cart04_front_temp														:= F_Temperature(TT_04_01, TT_04_01_offset);
cart04_front_temp_error 												:= TT_04_01_error OR iCount[6] < 30;
cart04_back_temp														:= F_Temperature(TT_04_03, TT_04_03_offset);
cart04_back_temp_error 													:= TT_04_03_Error OR iCount[7] < 30;
cart04_temp_front_calc(Error:= TT_04_01_error, Temp:= cart04_front_temp, Low:= sorbent_low_temp, High:= sorbent_high_temp, Total:= rTempTotal, Counter:= iTempCount);
cart04_temp_back_calc(Error:= TT_04_03_Error, Temp:= cart04_back_temp, Low:= sorbent_low_temp, High:= sorbent_high_temp, Total:= rTempTotal, Counter:= iTempCount);

cart05_front_temp														:= F_Temperature(TT_05_01, TT_05_01_offset);
cart05_front_temp_error 												:= TT_05_01_error OR iCount[8] < 30;
cart05_back_temp														:= F_Temperature(TT_05_03, TT_05_03_offset);
cart05_back_temp_error 													:= TT_05_03_Error OR iCount[9] < 30;
cart05_temp_front_calc(Error:= TT_05_01_error, Temp:= cart05_front_temp, Low:= sorbent_low_temp, High:= sorbent_high_temp, Total:= rTempTotal, Counter:= iTempCount);
cart05_temp_back_calc(Error:= TT_05_03_Error, Temp:= cart05_back_temp, Low:= sorbent_low_temp, High:= sorbent_high_temp, Total:= rTempTotal, Counter:= iTempCount);

cart06_front_temp														:= F_Temperature(TT_06_01, TT_06_01_offset);
cart06_front_temp_error 												:= TT_06_01_error OR iCount[10] < 30;
cart06_back_temp														:= F_Temperature(TT_06_03, TT_06_03_offset);
cart06_back_temp_error 													:= TT_06_03_Error OR iCount[11] < 30;
cart06_temp_front_calc(Error:= TT_06_01_error, Temp:= cart06_front_temp, Low:= sorbent_low_temp, High:= sorbent_high_temp, Total:= rTempTotal, Counter:= iTempCount);
cart06_temp_back_calc(Error:= TT_06_03_Error, Temp:= cart06_back_temp, Low:= sorbent_low_temp, High:= sorbent_high_temp, Total:= rTempTotal, Counter:= iTempCount);

cart07_front_temp														:= F_Temperature(TT_07_01, TT_07_01_offset);
cart07_front_temp_error 												:= TT_07_01_error OR iCount[12] < 30;
cart07_back_temp														:= F_Temperature(TT_07_03, TT_07_03_offset);
cart07_back_temp_error 													:= TT_07_03_Error OR iCount[13] < 30;
cart07_temp_front_calc(Error:= TT_07_01_error, Temp:= cart07_front_temp, Low:= sorbent_low_temp, High:= sorbent_high_temp, Total:= rTempTotal, Counter:= iTempCount);
cart07_temp_back_calc(Error:= TT_07_03_Error, Temp:= cart07_back_temp, Low:= sorbent_low_temp, High:= sorbent_high_temp, Total:= rTempTotal, Counter:= iTempCount);

cart08_front_temp														:= F_Temperature(TT_08_01, TT_08_01_offset);
cart08_front_temp_error 												:= TT_08_01_error OR iCount[14] < 30;
cart08_back_temp														:= F_Temperature(TT_08_03, TT_08_03_offset);
cart08_back_temp_error 													:= TT_08_03_Error OR iCount[15] < 30;
cart08_temp_front_calc(Error:= TT_08_01_error, Temp:= cart08_front_temp, Low:= sorbent_low_temp, High:= sorbent_high_temp, Total:= rTempTotal, Counter:= iTempCount);
cart08_temp_back_calc(Error:= TT_08_03_Error, Temp:= cart08_back_temp, Low:= sorbent_low_temp, High:= sorbent_high_temp, Total:= rTempTotal, Counter:= iTempCount);

cart09_front_temp														:= F_Temperature(TT_09_01, TT_09_01_offset);
cart09_front_temp_error 												:= TT_09_01_error OR iCount[16] < 30;
cart09_back_temp														:= F_Temperature(TT_09_03, TT_09_03_offset);
cart09_back_temp_error 													:= TT_09_03_Error OR iCount[17] < 30;
cart09_temp_front_calc(Error:= TT_09_01_error, Temp:= cart09_front_temp, Low:= sorbent_low_temp, High:= sorbent_high_temp, Total:= rTempTotal, Counter:= iTempCount);
cart09_temp_back_calc(Error:= TT_09_03_Error, Temp:= cart09_back_temp, Low:= sorbent_low_temp, High:= sorbent_high_temp, Total:= rTempTotal, Counter:= iTempCount);

cart10_front_temp														:= F_Temperature(TT_10_01, TT_10_01_offset);
cart10_front_temp_error 												:= TT_10_01_error OR iCount[18] < 30;
cart10_back_temp														:= F_Temperature(TT_10_03, TT_10_03_offset);
cart10_back_temp_error 													:= TT_10_03_Error OR iCount[19] < 30;
cart10_temp_front_calc(Error:= TT_10_01_error, Temp:= cart10_front_temp, Low:= sorbent_low_temp, High:= sorbent_high_temp, Total:= rTempTotal, Counter:= iTempCount);
cart10_temp_back_calc(Error:= TT_10_03_Error, Temp:= cart10_back_temp, Low:= sorbent_low_temp, High:= sorbent_high_temp, Total:= rTempTotal, Counter:= iTempCount);

cart11_front_temp														:= F_Temperature(TT_11_01, TT_11_01_offset);
cart11_front_temp_error 												:= TT_11_01_error OR iCount[20] < 30;
cart11_back_temp														:= F_Temperature(TT_11_03, TT_11_03_offset);
cart11_back_temp_error 													:= TT_11_03_Error OR iCount[21] < 30;
cart11_temp_front_calc(Error:= TT_11_01_error, Temp:= cart11_front_temp, Low:= sorbent_low_temp, High:= sorbent_high_temp, Total:= rTempTotal, Counter:= iTempCount);
cart11_temp_back_calc(Error:= TT_11_03_Error, Temp:= cart11_back_temp, Low:= sorbent_low_temp, High:= sorbent_high_temp, Total:= rTempTotal, Counter:= iTempCount);

cart12_front_temp														:= F_Temperature(TT_12_01, TT_12_01_offset);
cart12_front_temp_error 												:= TT_12_01_error OR iCount[22] < 30;
cart12_back_temp														:= F_Temperature(TT_12_03, TT_12_03_offset);
cart12_back_temp_error 													:= TT_12_03_Error OR iCount[23] < 30;
cart12_temp_front_calc(Error:= TT_12_01_error, Temp:= cart12_front_temp, Low:= sorbent_low_temp, High:= sorbent_high_temp, Total:= rTempTotal, Counter:= iTempCount);
cart12_temp_back_calc(Error:= TT_12_03_Error, Temp:= cart12_back_temp, Low:= sorbent_low_temp, High:= sorbent_high_temp, Total:= rTempTotal, Counter:= iTempCount);

sorbent_average_temp													:= SEL(iTempCount > 0, 0, rTempTotal / iTempCount);

FOR i:= 0 TO 23 DO
	iCount[i]															:= iCount[i] + 1;
	IF iCount[i] > 30 THEN
		iCount[i]														:= 30;
	END_IF
END_FOR

iHighTempCount															:= 0;
rMin																	:= u01.SP_minimum_reasonable_sorbent_TC_reading;
rMax																	:= u01.SP_maximum_reasonable_sorbent_TC_reading;
IF iInletAirSetpoint = 0 THEN
	rTempSP																:= m01.SP_vacuum_cooling_target_temperature;
ELSIF iInletAirSetpoint = 1 THEN
	rTempSP																:= m01.SP_maximum_inlet_air_temperature_during_adsorption;
ELSE
	rTempSP																:= m01.SP_maximum_sorbent_temperature_during_desorption;
END_IF

IF TT_01_01_Error OR cart01_front_temp < rMin OR cart01_front_temp > rMax THEN
	iCount[0]															:= 0;
ELSIF cart01_front_temp > rTempSP THEN
	iHighTempCount														:= iHighTempCount + 1;
END_IF 
IF TT_01_03_Error OR cart01_back_temp < rMin OR cart01_back_temp > rMax THEN
	iCount[1]															:= 0;
ELSIF cart01_back_temp > rTempSP THEN
	iHighTempCount														:= iHighTempCount + 1;
END_IF

IF TT_02_01_Error OR cart02_front_temp < rMin OR cart02_front_temp > rMax THEN
	iCount[2]															:= 0;
ELSIF cart02_front_temp > rTempSP THEN
	iHighTempCount														:= iHighTempCount + 1;
END_IF 
IF TT_02_03_Error OR cart02_back_temp < rMin OR cart02_back_temp > rMax THEN
	iCount[3]															:= 0;
ELSIF cart02_back_temp > rTempSP THEN
	iHighTempCount														:= iHighTempCount + 1;
END_IF

IF TT_03_01_Error OR cart03_front_temp < rMin OR cart03_front_temp > rMax THEN
	iCount[4]															:= 0;
ELSIF cart03_front_temp > rTempSP THEN
	iHighTempCount														:= iHighTempCount + 1;
END_IF 
IF TT_03_03_Error OR cart03_back_temp < rMin OR cart03_back_temp > rMax THEN
	iCount[5]															:= 0;
ELSIF cart03_back_temp > rTempSP THEN
	iHighTempCount														:= iHighTempCount + 1;
END_IF

IF TT_04_01_Error OR cart04_front_temp < rMin OR cart04_front_temp > rMax THEN
	iCount[6]															:= 0;
ELSIF cart04_front_temp > rTempSP THEN
	iHighTempCount														:= iHighTempCount + 1;
END_IF 
IF TT_04_03_Error OR cart04_back_temp < rMin OR cart04_back_temp > rMax THEN
	iCount[7]															:= 0;
ELSIF cart04_back_temp > rTempSP THEN
	iHighTempCount														:= iHighTempCount + 1;
END_IF

IF TT_05_01_Error OR cart05_front_temp < rMin OR cart05_front_temp > rMax THEN
	iCount[8]															:= 0;
ELSIF cart05_front_temp > rTempSP THEN
	iHighTempCount														:= iHighTempCount + 1;
END_IF 
IF TT_05_03_Error OR cart05_back_temp < rMin OR cart05_back_temp > rMax THEN
	iCount[9]															:= 0;
ELSIF cart05_back_temp > rTempSP THEN
	iHighTempCount														:= iHighTempCount + 1;
END_IF

IF TT_06_01_Error OR cart06_front_temp < rMin OR cart06_front_temp > rMax THEN
	iCount[10]															:= 0;
ELSIF cart06_front_temp > rTempSP THEN
	iHighTempCount														:= iHighTempCount + 1;
END_IF 
IF TT_06_03_Error OR cart06_back_temp < rMin OR cart06_back_temp > rMax THEN
	iCount[11]															:= 0;
ELSIF cart06_back_temp > rTempSP THEN
	iHighTempCount														:= iHighTempCount + 1;
END_IF

IF TT_07_01_Error OR cart07_front_temp < rMin OR cart07_front_temp > rMax THEN
	iCount[12]															:= 0;
ELSIF cart07_front_temp > rTempSP THEN
	iHighTempCount														:= iHighTempCount + 1;
END_IF 
IF TT_07_03_Error OR cart07_back_temp < rMin OR cart07_back_temp > rMax THEN
	iCount[13]															:= 0;
ELSIF cart07_back_temp > rTempSP THEN
	iHighTempCount														:= iHighTempCount + 1;
END_IF

IF TT_08_01_Error OR cart08_front_temp < rMin OR cart08_front_temp > rMax THEN
	iCount[14]															:= 0;
ELSIF cart08_front_temp > rTempSP THEN
	iHighTempCount														:= iHighTempCount + 1;
END_IF 
IF TT_08_03_Error OR cart08_back_temp < rMin OR cart08_back_temp > rMax THEN
	iCount[15]															:= 0;
ELSIF cart08_back_temp > rTempSP THEN
	iHighTempCount														:= iHighTempCount + 1;
END_IF

IF TT_09_01_Error OR cart09_front_temp < rMin OR cart09_front_temp > rMax THEN
	iCount[16]															:= 0;
ELSIF cart09_front_temp > rTempSP THEN
	iHighTempCount														:= iHighTempCount + 1;
END_IF 
IF TT_09_03_Error OR cart09_back_temp < rMin OR cart09_back_temp > rMax THEN
	iCount[17]															:= 0;
ELSIF cart09_back_temp > rTempSP THEN
	iHighTempCount														:= iHighTempCount + 1;
END_IF

IF TT_10_01_Error OR cart10_front_temp < rMin OR cart10_front_temp > rMax THEN
	iCount[18]															:= 0;
ELSIF cart10_front_temp > rTempSP THEN
	iHighTempCount														:= iHighTempCount + 1;
END_IF 
IF TT_10_03_Error OR cart10_back_temp < rMin OR cart10_back_temp > rMax THEN
	iCount[19]															:= 0;
ELSIF cart10_back_temp > rTempSP THEN
	iHighTempCount														:= iHighTempCount + 1;
END_IF

IF TT_11_01_Error OR cart11_front_temp < rMin OR cart11_front_temp > rMax THEN
	iCount[20]															:= 0;
ELSIF cart11_front_temp > rTempSP THEN
	iHighTempCount														:= iHighTempCount + 1;
END_IF 
IF TT_11_03_Error OR cart11_back_temp < rMin OR cart11_back_temp > rMax THEN
	iCount[21]															:= 0;
ELSIF cart11_back_temp > rTempSP THEN
	iHighTempCount														:= iHighTempCount + 1;
END_IF

IF TT_12_01_Error OR cart12_front_temp < rMin OR cart12_front_temp > rMax THEN
	iCount[22]															:= 0;
ELSIF cart12_front_temp > rTempSP THEN
	iHighTempCount														:= iHighTempCount + 1;
END_IF 
IF TT_12_03_Error OR cart12_back_temp < rMin OR cart12_back_temp > rMax THEN
	iCount[23]															:= 0;
ELSIF cart12_back_temp > rTempSP THEN
	iHighTempCount														:= iHighTempCount + 1;
END_IF

IF iInletAirSetpoint = 0 THEN
	vacuum_cooling_high_temp_count										:= iHighTempCount;
ELSIF iInletAirSetpoint = 1 THEN
	adsorption_high_temp_count											:= iHighTempCount;
ELSE
	desorption_high_temp_count											:= iHighTempCount;
END_IF
iInletAirSetpoint														:= SEL(iInletAirSetpoint = 2, iInletAirSetpoint + 1, 0);;
END_ACTION

END_FUNCTION_BLOCK

// ---- POUs/Function_Blocks/FB_Temperature.TcPOU
FUNCTION_BLOCK FB_Temperature
VAR_INPUT
	Error																: BOOL;
	Temp																: REAL;
	Low																	: REFERENCE TO REAL;
	High																: REFERENCE TO REAL;
	Total																: REFERENCE TO REAL;
	Counter																: REFERENCE TO INT;
END_VAR
VAR
END_VAR

// Phase 0 - FB_Temperature
// Rev 1.0 - April 25, 2024

IF NOT Error THEN
	Low																	:= F_LowestReal(Temp, Low);
	High																:= F_HighestReal(Temp, High, 0, 0);
	Total																:= Total + Temp;
	Counter																:= Counter + 1;
END_IF

END_FUNCTION_BLOCK

// ---- POUs/Functions/F_LowestReal.TcPOU
FUNCTION F_LowestReal : REAL
VAR_INPUT
	Value1																: REAL;
	Value2																: REAL;
END_VAR
VAR
END_VAR

// F_LowerValue
// Rev 1.0 - March 14, 2024

F_LowestReal															:= SEL(Value1 < Value2, Value2, Value1);

END_FUNCTION

// ---- POUs/Functions/F_Temperature.TcPOU
FUNCTION F_Temperature : REAL
VAR_INPUT
	Input																: INT;
	Offset																: REAL;
END_VAR
VAR
END_VAR

// F_Temperature
// Rev 1.0 - December 28, 2023

F_Temperature															:= INT_TO_REAL(Input) / 10.0 + Offset;

END_FUNCTION

// ---- POUs/Functions/F_AnalogIn.TcPOU
FUNCTION F_AnalogIn : REAL
VAR_INPUT
	Input																: INT;
	Low																	: REAL;
	High																: REAL;
	Minimum																: REAL;
	Offset																: REAL;
END_VAR
VAR
	Value											: REAL;
END_VAR

// F_AnalogIn
// Rev 1.0 - December 28, 2023

Value																	:= ((High - Low) / 32767.0) * INT_TO_REAL(Input) + Low;		// Determine output based on scale
Value																	:= Value + Offset;											// Adjust for any user offset
F_AnalogIn																:= SEL(ABS(Value) > Minimum, 0, Value);						// Value must be above (or below, if negative) minimum or zero is returned

END_FUNCTION

// ---- POUs/Module_01/P_M01.TcPOU
PROGRAM P_M01
VAR PERSISTENT
	udiCycleCountRS01													: DINT;
	udiCycleCountRS02													: DINT;
	udiCycleCountRS03													: DINT;
END_VAR
VAR
	m																	: Module;
	sCycleModeRS01														: STRING	:= '';
	sCycleModeRS02														: STRING	:= '';
	sCycleModeRS03														: STRING	:= '';
	iRS01CyclesToRun													: INT;
	iRS02CyclesToRun													: INT;
	iRS03CyclesToRun													: INT;
	iLength																: INT;
	iReactorSetToActivate												: INT;
	iRS01Count															: INT;
	iRS02Count															: INT;
	iRS03Count															: INT;
	rtrigStart															: R_TRIG;
	
	bRSProcess															: BOOL;
	bRSManual															: BOOL;
	bRS01																: BOOL;
	bRS02																: BOOL;
	bRS03																: BOOL;
	bRS01Selected														: BOOL;
	bRS02Selected														: BOOL;
	bRS03Selected														: BOOL;
	bRSTimer															: BOOL;
	bStarted															: BOOL;
	bReactorSetSelected													: BOOL;
	
	rtrigRS01StartNextRS												: R_TRIG;
	rtrigRS02StartNextRS												: R_TRIG;
	rtrigRS03StartNextRS												: R_TRIG;
	rtrigRS01Restart													: R_TRIG;
	rtrigRS02Restart													: R_TRIG;
	rtrigRS03Restart													: R_TRIG;
	rtrigRS01Done														: R_TRIG;
	rtrigRS02Done														: R_TRIG;
	rtrigRS03Done														: R_TRIG;
	rtrigRS01Offline													: R_TRIG;
	rtrigRS02Offline													: R_TRIG;
	rtrigRS03Offline													: R_TRIG;
	
	tonRSTimer															: TON;
	
	fb_Condensate_From_Cooling_And_Purge_Lines_Pump						: FB_Digital_Out();
	
	rtrigCPDrainLSHOn													: R_TRIG;
	tonCPDrainErrorOn													: TON;
	tonCPDrainErrorOff													: TON;
	bCPDrainError														: BOOL;
	
	rMinPressureSP														: REAL; 
	rMaxPressureSP														: REAL;
	
	bCondensateFlowError												: BOOL;
	bSteamManifoldLinePresError											: BOOL;
	bSteamTempNearRS01Error												: BOOL;
	bSteamTempNearRS03Error												: BOOL;
	bCondensateTempError												: BOOL;
	
	sModuleError														: STRING;
	
	evac_service_acked													: BOOL;
	steam_service_acked													: BOOL;
	
	deadair_pump_req													: ST_Util_Service_Req;
	steam_system_req													: ST_Util_Service_Req;
	
	fb_util_service_ctrl 												: FB_Util_Service_Control;
	
	evac_service_assigned												: ARRAY[1..rs_count] OF BOOL;
	evac_service_req													: ARRAY[1..rs_count] OF BOOL;
	
	steam_service_assigned												: ARRAY[1..rs_count] OF BOOL;
	steam_service_req													: ARRAY[1..rs_count] OF BOOL;
	
	idx_rs																: INT;
END_VAR

// Phase 0 - P_M01
// Rev 1.0 - May 1, 2024

m01.condensate_flow														:= F_AnalogIn(m01.FT_02, m01.condensate_flow_low, m01.condensate_flow_high, m01.condensate_flow_min, m01.condensate_flow_offset);
m.condensate_flow														:= m01.condensate_flow;
m.condensate_flow_error													:= m01.condensate_flow_error AND NOT _CondensateFlowOff;
bCondensateFlowError													:= P_Alarms.M_Check_Error(m01.condensate_flow_error, bCondensateFlowError, _M01, gsCondesateFlowSensorError, gsProcessCannotRun);

m01.steam_manifold_line_pres											:= F_AnalogIn(m01.PT_02, m01.steam_manifold_line_pres_low, m01.steam_manifold_line_pres_high, m01.steam_manifold_line_pres_min, m01.steam_manifold_line_pres_offset);
m.steam_manifold_line_pres												:= m01.steam_manifold_line_pres;
m.steam_manifold_line_pres_error										:= m01.steam_manifold_line_pres_error AND NOT _SteamManifoldLinePresOff;
bSteamManifoldLinePresError												:= P_Alarms.M_Check_Error(m01.steam_manifold_line_pres_error, bSteamManifoldLinePresError, _M01, gsSteamManifoldLinePresSensorError, gsProcessCannotRun);

m.condensate_from_cooling_and_purge_lines_lsl							:= m01.condensate_from_cooling_and_purge_lines_lsl;
m.condensate_from_cooling_and_purge_lines_lsh							:= m01.condensate_from_cooling_and_purge_lines_lsh;

fb_Condensate_From_Cooling_And_Purge_Lines_Pump(Input1:= m01.condensate_from_cooling_and_purge_lines_pump, Input2:= m.condensate_from_cooling_and_purge_lines_pump, Output=> m01.P_02);
m01.condensate_from_cooling_and_purge_lines_pump_cmd_status				:= m01.P_02;

m01.steam_temp_near_rs1													:= F_Temperature(m01.TT_10, m01.steam_temp_near_rs1_offset);
m.steam_temp_near_rs1													:= m01.steam_temp_near_rs1;
m.steam_temp_near_rs1_error												:= m01.steam_temp_near_rs1_error AND NOT _SteamTempNearRS01Off;
bSteamTempNearRS01Error													:= P_Alarms.M_Check_Error(m.steam_temp_near_rs1_error, bSteamTempNearRS01Error, _M01, gsSteamTempNearRS01SensorError, gsProcessCannotRun);

m01.steam_temp_near_rs3													:= F_Temperature(m01.TT_11, m01.steam_temp_near_rs3_offset);
m.steam_temp_near_rs3													:= m01.steam_temp_near_rs3;
m.steam_temp_near_rs3_error												:= m01.steam_temp_near_rs3_error AND NOT _SteamTempNearRS03Off;
bSteamTempNearRS03Error													:= P_Alarms.M_Check_Error(m.steam_temp_near_rs3_error, bSteamTempNearRS03Error, _M01, gsSteamTempNearRS03SensorError, gsProcessCannotRun);

m01.condensate_temp														:= F_Temperature(m01.TT_12, m01.condensate_temp_offset);
m.condensate_temp														:= m01.condensate_temp;
m.condensate_temp_error													:= m01.condensate_temp_error AND NOT _CondensateTempOff;
bCondensateTempError													:= P_Alarms.M_Check_Error(m.condensate_temp_error, bCondensateTempError, _M01, gsCondensateTempSensorError, gsProcessCannotRun);

// Ignore if < 2 amps 
m01.l1_current															:= SEL(m01.IT_01 > _CURRENT_MODULE_FACTOR *2,0,F_IEConvert(m01.IT_01, _CURRENT_MODULE_FACTOR));
m01.l2_current															:= SEL(m01.IT_02 > _CURRENT_MODULE_FACTOR *2,0,F_IEConvert(m01.IT_02, _CURRENT_MODULE_FACTOR));
m01.l3_current															:= SEL(m01.IT_03 > _CURRENT_MODULE_FACTOR *2,0,F_IEConvert(m01.IT_03, _CURRENT_MODULE_FACTOR));
m01.l1_voltage															:= F_IEConvert(m01.VT_01, _VOLTAGE_480_FACTOR);
m01.l2_voltage															:= F_IEConvert(m01.VT_02, _VOLTAGE_480_FACTOR);
m01.l3_voltage															:= F_IEConvert(m01.VT_03, _VOLTAGE_480_FACTOR);

A_Drain_Condensate_Product_Cooling_Lines();

P_M01_RS01();
P_M01_RS02();
P_M01_RS03();

rMinPressureSP															:= m01.SP_ambient_pressure - (m01.SP_percent_of_ambient_pressure / 100 * m01.SP_ambient_pressure); 
rMaxPressureSP															:= m01.SP_ambient_pressure + (m01.SP_percent_of_ambient_pressure / 100 * m01.SP_ambient_pressure);

sModuleError															:= SEL(bSteamManifoldLinePresError, sModuleError, gsSteamManifoldLinePresSensorError);		// Start up error
sModuleError															:= SEL(bSteamTempNearRS01Error, sModuleError, gsSteamTempNearRS01SensorError);				// Start up error
sModuleError															:= SEL(bSteamTempNearRS03Error, sModuleError, gsSteamTempNearRS03SensorError);				///! Not in prestart check
sModuleError															:= SEL(bCondensateTempError, sModuleError, gsCondensateTempSensorError);					///! Not in prestart check
sModuleError															:= SEL(bCondensateFlowError, '', gsCondesateFlowSensorError);								///! Not in prestart check
 
A_AutoMode();

ACTION A_AutoMode:
// Phase 0 - P_M01.A_AutoMode
// Rev 1.0 - May 11, 2024

IF m01.tb_Stop_Process OR P_M01_RS01.utility_error OR P_M01_RS02.utility_error OR P_M01_RS03.utility_error THEN 			// Stop all processes from HMI or if utility error occurs
	u01.shutdown_process												:= TRUE;
//	IF m01.tb_Auto_Mode_On THEN
	P_M01_RS01.stop_rs_automode										:= TRUE;
	P_M01_RS02.stop_rs_automode										:= TRUE;
	P_M01_RS03.stop_rs_automode										:= TRUE;
//	END_IF
	bRSProcess															:= FALSE;
	m01.tb_Stop_Process													:= FALSE;
END_IF

IF m01.tb_Cancel_Cycle OR P_M01_RS01.cancel_all_reactor_sets OR P_M01_RS02.cancel_all_reactor_sets OR P_M01_RS03.cancel_all_reactor_sets THEN																									// Complete current cycles then stop
	iRS01CyclesToRun													:= SEL(m01_rs1.tb_Process_Running, iRS01Count, iRS01Count + 1);
	iRS02CyclesToRun													:= SEL(m01_rs2.tb_Process_Running, iRS02Count, iRS02Count + 1);
	iRS03CyclesToRun													:= SEL(m01_rs3.tb_Process_Running, iRS03Count, iRS03Count + 1);
	bRS01																:= SEL(iRS01Count >= iRS01CyclesToRun, bRS01, FALSE);
	bRS02																:= SEL(iRS02Count >= iRS02CyclesToRun, bRS02, FALSE);
	bRS03																:= SEL(iRS03Count >= iRS03CyclesToRun, bRS03, FALSE);
	m01.tb_Cancel_Cycle													:= FALSE;
END_IF

A_AutoMode_RS01();
A_AutoMode_RS02();
A_AutoMode_RS03();

bReactorSetSelected														:= m01.SP_include_reactor_set_1_in_process OR m01.SP_include_reactor_set_2_in_process OR m01.SP_include_reactor_set_3_in_process;
IF m01.ts_Cycle_Mode <> '' AND (sModuleError <> '' OR P_U01.sUtilityError <> '' OR m01.SP_desired_cycle_count = 0 OR NOT bReactorSetSelected) THEN		// Don't allow cycle if moodule or utility error occured, cycle count is zero or no reactor sets are selected
	IF sModuleError <> '' THEN
		P_Alarms.M_Add_Alarm(_M01, sModuleError, gsProcessCannotRun);
	ELSIF P_U01.sUtilityError  <> '' THEN
		P_Alarms.M_Add_Alarm(_U01, P_U01.sUtilityError, gsProcessCannotRun);
	ELSIF m01.SP_desired_cycle_count = 0 THEN
		P_Alarms.M_Add_Alarm(_U01, gsDesiredCycleCountError, gsProcessCannotRun);
	ELSE
		P_Alarms.M_Add_Alarm(_U01, gsNoReactorSetsSelected, gsProcessCannotRun);
	END_IF
	m01.ts_Cycle_Mode													:= '';
END_IF

iLength																	:= LEN(m01.ts_Cycle_Mode);							// Start process in this order '6745' (Evap, Desorp, Repres, Adsorp)
rtrigStart(CLK:= iLength > 0);
IF rtrigStart.Q THEN
	gsCycleMode															:= m01.ts_Cycle_Mode;
	m01.ts_Cycle_Mode													:= '';
	iRS01CyclesToRun													:= m01.SP_desired_cycle_count;
	iRS02CyclesToRun													:= m01.SP_desired_cycle_count;
	iRS03CyclesToRun													:= m01.SP_desired_cycle_count;
	bRS01																:= m01.SP_include_reactor_set_1_in_process;			// Get active reactors
	bRS02																:= m01.SP_include_reactor_set_2_in_process;                         
	bRS03																:= m01.SP_include_reactor_set_3_in_process;
	IF iLength = 1 THEN																										// Single process selected
		m01.tb_Auto_Mode_On												:= FALSE;
		bRSManual														:= STRING_TO_INT(gsCycleMode) >= eRepressurization AND STRING_TO_INT(gsCycleMode) <= eDesorption;
	ELSE
		iReactorSetToActivate											:= SEL(bRS01, SEL(bRS02, SEL(bRS03, 0, 3), 2), 1);	// Determine which reactor set to start
        IF iReactorSetToActivate > 0 THEN																					// Start process if at least one reactor set is selected              
			bRS01Selected												:= bRS01;
			bRS02Selected												:= bRS02;
			bRS03Selected												:= bRS03;
			m01_rs1.ti_Cycle_Count										:= 0;												// Completed cycles
			m01_rs2.ti_Cycle_Count										:= 0;
			m01_rs3.ti_Cycle_Count										:= 0;
			iRS01Count													:= 0;												// Attempted cycles
			iRS02Count													:= 0;
			iRS03Count													:= 0;
			m01.tb_Auto_Mode_On											:= TRUE;
			bRSProcess													:= TRUE;
		END_IF
	END_IF

	
END_IF

IF bRSManual THEN
	
	sCycleModeRS01														:= SEL(bRS01, sCycleModeRS01, gsCycleMode);
	sCycleModeRS02														:= SEL(bRS02, sCycleModeRS02, gsCycleMode);
	sCycleModeRS03														:= SEL(bRS03, sCycleModeRS03, gsCycleMode);
	bRSManual															:= FALSE;
	
ELSIF bRSProcess THEN
	
	rtrigRS01Done(CLK:= P_M01_RS01.reactor_done);
	IF rtrigRS01Done.Q THEN
		sCycleModeRS01													:= '';												// Turn off cycle
		iRS01Count														:= iRS01Count + 1;									// This counter increments regardless of reactor status if long as reactor was selected
		IF iRS01Count >= iRS01CyclesToRun THEN
			bRS01														:= FALSE;
		END_IF
		IF m01_rs1.tb_Process_Complete THEN 																				// Increment these counters once a valid cycle has run
			m01_rs1.ti_Cycle_Count										:= m01_rs1.ti_Cycle_Count + 1;
			udiCycleCountRS01											:= udiCycleCountRS01 + 1;
			m01_rs1.ti_Total_Cycle_Count								:= udiCycleCountRS01;
		END_IF
	END_IF
	
	rtrigRS02Done(CLK:= P_M01_RS02.reactor_done);
	IF rtrigRS02Done.Q THEN
		sCycleModeRS02													:= '';
		iRS02Count														:= iRS02Count + 1;
		IF iRS02Count >= iRS02CyclesToRun THEN
			bRS02														:= FALSE;
		END_IF
		IF m01_rs2.tb_Process_Complete THEN 
			m01_rs2.ti_Cycle_Count										:= m01_rs2.ti_Cycle_Count + 1;
			udiCycleCountRS02											:= udiCycleCountRS02 + 1;
			m01_rs2.ti_Total_Cycle_Count								:= udiCycleCountRS02;
		END_IF
	END_IF
	
	rtrigRS03Done(CLK:= P_M01_RS03.reactor_done);
	IF rtrigRS03Done.Q THEN
		sCycleModeRS03													:= '';
		iRS03Count														:= iRS03Count + 1;
		IF iRS03Count >= iRS03CyclesToRun THEN
			bRS03														:= FALSE;
		END_IF
		IF m01_rs3.tb_Process_Complete THEN 
			m01_rs3.ti_Cycle_Count										:= m01_rs3.ti_Cycle_Count + 1;
			udiCycleCountRS03											:= udiCycleCountRS03 + 1;
			m01_rs3.ti_Total_Cycle_Count								:= udiCycleCountRS03;
		END_IF
	END_IF

	bRSTimer															:= TRUE;
	IF tonRSTimer.Q OR NOT bStarted THEN
		IF iReactorSetToActivate = 1 THEN
			IF NOT m01_rs1.tb_Process_Running THEN
				sCycleModeRS01											:= SEL(bRS01, '0', gsCycleMode);
				iReactorSetToActivate									:= 2;
				bRSTimer												:= NOT bRS01;
			END_IF
		ELSIF iReactorSetToActivate = 2 THEN
			IF NOT m01_rs2.tb_Process_Running THEN
				sCycleModeRS02											:= SEL(bRS02, '0', gsCycleMode);
				iReactorSetToActivate									:= 3;
				bRSTimer												:= NOT bRS02;
			END_IF
		ELSIF iReactorSetToActivate = 3 THEN
			IF NOT m01_rs3.tb_Process_Running THEN
				sCycleModeRS03											:= SEL(bRS03, '0', gsCycleMode);
				iReactorSetToActivate									:= 1;
				bRSTimer												:= NOT bRS03;
			END_IF
		END_IF
	END_IF
	IF NOT bRS01 AND NOT bRS02 AND NOT bRS03 THEN																				// Stop process when all reactor sets are done
		iReactorSetToActivate											:= 0;
		P_M01_RS01.stop_rs_automode										:= TRUE;
		P_M01_RS02.stop_rs_automode										:= TRUE;
		P_M01_RS03.stop_rs_automode										:= TRUE;
		bRSTimer														:= FALSE;
		bRSProcess														:= FALSE;
	END_IF
	bStarted															:= TRUE;
ELSE
//	u01.write_persistent_data											:= TRUE;
	sCycleModeRS01														:= '';
	sCycleModeRS02														:= '';
	sCycleModeRS03														:= '';
	bRS01																:= FALSE;
	bRS02																:= FALSE;
	bRS03																:= FALSE;
	giEvacuationErrorRS													:= 0;
	bStarted															:= FALSE;
	m01.tb_Auto_Mode_On													:= FALSE;
	
END_IF

// ========= Uitilities Service Request =========

//evac_service_acked := P_M01_RS01.fb_RS.Evac_Service_Req OR P_M01_RS02.fb_RS.Evac_Service_Req OR P_M01_RS03.fb_RS.Evac_Service_Req;

A_BOP_Services();


m01_rs1.cycle_stage														:= SEL(bRS01 AND gsCycleStage <> '', gsM01RS01CycleStage, gsCycleStage);
m01_rs2.cycle_stage														:= SEL(bRS02 AND gsCycleStage <> '', gsM01RS02CycleStage, gsCycleStage);
m01_rs3.cycle_stage														:= SEL(bRS03 AND gsCycleStage <> '', gsM01RS03CycleStage, gsCycleStage);

tonRSTimer(IN:= bRSTimer, PT:= REAL_TO_TIME(m01.SP_cycle_start_offset_duration * _MINUTES));
END_ACTION

ACTION A_AutoMode_RS01:
// Phase 0 - P_M01.A_AutoMode_RS01
// Rev 1.0 - May 10, 2024

rtrigRS01Restart(CLK:= m01.SP_include_reactor_set_1_in_process);
IF rtrigRS01Restart.Q THEN
	IF m01.tb_Auto_Mode_On AND NOT bRS01Selected THEN 
		m01.SP_include_reactor_set_1_in_process							:= FALSE;
	ELSE
		bRS01															:= TRUE;
		P_M01_RS01.clear_rs_pause										:= TRUE;
	END_IF
END_IF

IF P_M01_RS01.stop_rs_automode THEN
	m01.SP_include_reactor_set_1_in_process								:= FALSE;
	bRS01Selected														:= FALSE;
END_IF

rtrigRS01Offline(CLK:= NOT m01.SP_include_reactor_set_1_in_process);
IF rtrigRS01Offline.Q THEN
	bRS01																:= FALSE;
END_IF

IF P_M01_RS01.cancel_reactor_set THEN
	iRS01CyclesToRun													:= SEL(m01_rs1.tb_Process_Running, iRS01Count, iRS01Count + 1);
END_IF
END_ACTION

ACTION A_AutoMode_RS02:
// Phase 0 - P_M01.A_AutoMode_RS02
// Rev 1.0 - May 10, 2024

rtrigRS02Restart(CLK:= m01.SP_include_reactor_set_2_in_process);
IF rtrigRS02Restart.Q THEN
	IF m01.tb_Auto_Mode_On AND NOT bRS02Selected THEN
		m01.SP_include_reactor_set_2_in_process							:= FALSE;
	ELSE
		bRS02															:= TRUE;
		P_M01_RS02.clear_rs_pause										:= TRUE;
	END_IF
END_IF

IF P_M01_RS02.stop_rs_automode THEN
	m01.SP_include_reactor_set_2_in_process								:= FALSE;
	bRS02Selected														:= FALSE;
END_IF

rtrigRS02Offline(CLK:= NOT m01.SP_include_reactor_set_2_in_process);
IF rtrigRS02Offline.Q THEN
	bRS02																:= FALSE;
END_IF

IF P_M01_RS02.cancel_reactor_set THEN
	iRS02CyclesToRun													:= SEL(m01_rs2.tb_Process_Running, iRS02Count, iRS02Count + 1);
END_IF
END_ACTION

ACTION A_AutoMode_RS03:
// Phase 0 - P_M01.A_AutoMode_RS03
// Rev 1.0 - May 10, 2024

rtrigRS03Restart(CLK:= m01.SP_include_reactor_set_3_in_process);
IF rtrigRS03Restart.Q THEN
	IF m01.tb_Auto_Mode_On AND NOT bRS03Selected THEN
		m01.SP_include_reactor_set_3_in_process							:= FALSE;
	ELSE
		bRS03															:= TRUE;
		P_M01_RS03.clear_rs_pause										:= TRUE;
	END_IF
END_IF

IF P_M01_RS03.stop_rs_automode THEN
	m01.SP_include_reactor_set_3_in_process								:= FALSE;
	bRS03Selected														:= FALSE;
END_IF

rtrigRS03Offline(CLK:= NOT m01.SP_include_reactor_set_3_in_process);
IF rtrigRS03Offline.Q THEN
	bRS03																:= FALSE;
END_IF

IF P_M01_RS03.cancel_reactor_set THEN
	iRS03CyclesToRun													:= SEL(m01_rs3.tb_Process_Running, iRS03Count, iRS03Count + 1);
END_IF
END_ACTION

ACTION A_BOP_Services:

FOR idx_rs := 1 TO rs_count DO 
	evac_service_assigned[idx_rs] := fb_util_service_ctrl.RSs_ServiceAssiged(i_rs_number := idx_rs, i_assigned_rs_list := fb_util_service_ctrl.dead_air_pump.assigned_rs_number);
	steam_service_assigned[idx_rs] := fb_util_service_ctrl.RSs_ServiceAssiged(i_rs_number := idx_rs, i_assigned_rs_list := fb_util_service_ctrl.steam_system.assigned_rs_number);
	IF idx_rs = 1 THEN
		fb_util_service_ctrl.i_deadair_pump_req := P_M01_RS01.fb_RS.Evac_Service_Req;
		fb_util_service_ctrl.i_steam_system_req := P_M01_RS01.fb_RS.Steam_Service_Req;
	ELSIF idx_rs = 2 THEN
		fb_util_service_ctrl.i_deadair_pump_req := P_M01_RS02.fb_RS.Evac_Service_Req;
		fb_util_service_ctrl.i_steam_system_req := P_M01_RS02.fb_RS.Steam_Service_Req;
	ELSIF idx_rs = 3 THEN
		fb_util_service_ctrl.i_deadair_pump_req := P_M01_RS03.fb_RS.Evac_Service_Req;
		fb_util_service_ctrl.i_steam_system_req := P_M01_RS03.fb_RS.Steam_Service_Req;
	END_IF
	fb_util_service_ctrl.Services_Handler(i_rs_number_service_req := idx_rs);
END_FOR


fb_util_service_ctrl();
END_ACTION

ACTION A_Drain_Condensate_Product_Cooling_Lines:
// Phase 0 - P_M01.A_Drain_Condensate_Product_Cooling_Lines
// Rev 1.0 - March 4, 2024

IF gbDrainageOn THEN
	IF (u01.purge_product_line_pres < u01.SP_drainage_function_cutoff_pressure) OR
		(m01_rs1.purge_valve_closed AND m01_rs1.cooling_valve_closed AND m01_rs2.purge_valve_closed AND m01_rs2.cooling_valve_closed AND m01_rs3.purge_valve_closed AND m01_rs3.cooling_valve_closed) THEN
		m.condensate_from_cooling_and_purge_lines_pump					:= FALSE;
	ELSE
		IF m.condensate_from_cooling_and_purge_lines_lsh THEN
			m.condensate_from_cooling_and_purge_lines_pump				:= TRUE;
		END_IF
		IF NOT m.condensate_from_cooling_and_purge_lines_lsl THEN
			m.condensate_from_cooling_and_purge_lines_pump				:= FALSE;
		END_IF
	END_IF
	
	rtrigCPDrainLSHOn(CLK:= tonCPDrainErrorOn.Q);
	IF rtrigCPDrainLSHOn.Q THEN
		P_Alarms.M_Add_Alarm(_M01, gsCondensateProductDrainError, gsProcessStopsAtEOC);
		m.condensate_from_cooling_and_purge_lines_pump					:= FALSE;
		bCPDrainError													:= TRUE;
		m01.tb_Cancel_Cycle												:= TRUE;											// Complete current cycles
	END_IF
	tonCPDrainErrorOn(IN:= m.condensate_from_cooling_and_purge_lines_lsh AND NOT bCPDrainError, PT:= _DRAIN_TIME);
	
	IF tonCPDrainErrorOff.Q THEN
		bCPDrainError													:= FALSE;
	END_IF
	tonCPDrainErrorOff(IN:= NOT m.condensate_from_cooling_and_purge_lines_lsh AND bCPDrainError, PT:= _DRAIN_TIME);
END_IF
END_ACTION

END_PROGRAM

// ---- POUs/Function_Blocks/FB_Util_Service_Control.TcPOU
FUNCTION_BLOCK FB_Util_Service_Control

VAR_INPUT	

	i_deadair_pump_req			: BOOL;
	i_steam_system_req			: BOOL;
	
END_VAR

VAR_OUTPUT
	o_bop_error_estop					: BOOL;
END_VAR

VAR

	deadair_pump_req		: ST_Util_Service_Req;
	steam_system_req		: ST_Util_Service_Req;

	dead_air_pump	: FB_Util_Service(shared_rs_count := 1,	module_rs_constrain := FALSE, manual_control_only := FALSE);
	steam_system 	: FB_Util_Service(shared_rs_count := 1, module_rs_constrain := FALSE,  manual_control_only := FALSE);
	
END_VAR


o_bop_error_estop := P_U01.u.utility_error <> '';


IF o_bop_error_estop  THEN
	  Clear_Services_Queue();	 
END_IF

METHOD Clear_Services_Queue : BOOL
VAR_INPUT
END_VAR

dead_air_pump.Clear_RS_Queue();
steam_system.Clear_RS_Queue();
END_METHOD

METHOD RSs_ServiceAssiged : BOOL
VAR_INPUT
	i_rs_number : INT;
	i_assigned_rs_list : ARRAY[1..rs_count] OF UINT; 
END_VAR
VAR
	idx_rs : INT;
END_VAR
// TRUE if a RS is assigned to an utilities service 

FOR idx_rs := 1 TO rs_count DO 
	IF i_rs_number = TO_INT(i_assigned_rs_list[idx_rs]) THEN
		RSs_ServiceAssiged := TRUE;
		EXIT;
	END_IF
END_FOR
END_METHOD

METHOD Services_Handler : BOOL
VAR_INPUT
	i_rs_number_service_req		: UINT;

END_VAR
// Services FB calls
	

deadair_pump_req.request_cmd := i_deadair_pump_req;
deadair_pump_req.rs_number := i_rs_number_service_req;
				 
dead_air_pump( i_service_req := deadair_pump_req, 
			   i_fault_req := o_bop_error_estop, 
			   o_activeQueue_number => m01.dispatch_active_queue_dead_pump,	
			   o_passiveQueue_number => m01.dispatch_passive_queue_dead_pump,
			  );
			   
			   
steam_system_req.request_cmd := i_steam_system_req;
steam_system_req.rs_number := i_rs_number_service_req;			   

steam_system(i_service_req := steam_system_req, 
			i_fault_req := o_bop_error_estop,
			o_activeQueue_number => m01.dispatch_active_queue_steam_pump,
			o_passiveQueue_number => m01.dispatch_passive_queue_steam_pump,
			);
END_METHOD

END_FUNCTION_BLOCK

// ---- POUs/Function_Blocks/FB_Util_Service.TcPOU
FUNCTION_BLOCK FB_Util_Service

VAR_INPUT
	i_service_req			: ST_Util_Service_Req;
	i_fault_req				: BOOL;   // fault request from additional services
END_VAR

VAR_OUTPUT
	o_service_sts 			: ST_Util_Service_Sts;
	o_bService_sts			: BYTE;
	o_activeQueue_number	:  ARRAY[1..rs_count] OF UINT;
	o_passiveQueue_number	:  ARRAY[1..rs_count] OF UINT;
END_VAR

VAR
	shared_rs_count  		: INT;     // max number of rs to be assigned to the util service
	module_rs_constrain		: BOOL;		// same module assignment constrain
	manual_control_only		: BOOL;		// manual control only 
	
	service_req 			: BOOL;
	service_req_dispatcher	: BOOL;
		
	fb_dispatcher 			: FB_Service_Dispatcher;
	
END_VAR


// Dispatcher call for adding the RSs to the services queue
  
IF  i_fault_req THEN 
	
	Clear_RS_Queue();
	
ELSE
	
// manage the rs assignment queue based on request form reactor set controller, max number of RSs shared by the service and the number of RSs whithin the same module that can sahre the same service 

	fb_dispatcher( i_service_req := i_service_req,
				   i_shared_rs := shared_rs_count,
				   i_rs_module_constrain := module_rs_constrain, 
				   o_service_req => service_req_dispatcher,
				   o_assigned_rs_number=>o_activeQueue_number, 
				   o_passiveQueue_number => o_passiveQueue_number);
	   
	
END_IF

PROPERTY assigned_rs_number : ARRAY[1..rs_count] OF UINT
GET

assigned_rs_number := fb_dispatcher.o_assigned_rs_number;
END_GET
END_PROPERTY

METHOD Clear_RS_Queue : BOOL
fb_dispatcher.Clear_Queue();
END_METHOD

METHOD FB_init : BOOL
VAR_INPUT
	bInitRetains 		: BOOL; // if TRUE, the retain variables are initialized (warm start / cold start)
	bInCopyCode 		: BOOL;  // if TRUE, the instance afterwards gets moved into the copy code (online change)
	shared_rs_count  	: UINT;
	module_rs_constrain	: BOOL;
	manual_control_only : BOOL;
END_VAR
THIS^.shared_rs_count := shared_rs_count;
THIS^.module_rs_constrain := module_rs_constrain;
THIS^.manual_control_only := manual_control_only;
END_METHOD

END_FUNCTION_BLOCK

// ---- POUs/Function_Blocks/FB_Service_Dispatcher.TcPOU
FUNCTION_BLOCK FB_Service_Dispatcher
VAR_INPUT
	i_service_req 			: ST_Util_Service_Req;
	i_shared_rs 			: INT;		  // max number of reactor sets  the util service can be shared by 
	i_rs_module_constrain  	: BOOL;       // true if the reactors sets cannot be par of the same module
END_VAR
VAR_OUTPUT
	o_service_req			: BOOL;  // on/off request to utilities 
	o_assigned_rs_number	: ARRAY[1..rs_count] OF UINT; // rs number that has been assigned to a service 
	o_passiveQueue_number	: ARRAY[1..rs_count] OF UINT;
END_VAR
VAR
	service_req_queue		: ARRAY [1..rs_count] OF ST_Service_Assigned_Sts;
	idx_queue				: INT;
	idx_queue_update		: INT;
	trig_service_assign		: R_TRIG;
	trig_service_release	: R_TRIG;
	
	service_assign			: BOOL;
	service_release			: BOOL;
	
	rs_same_module			: BOOL;
END_VAR

// Add to queue 

FOR idx_queue := 1 TO rs_count DO
	IF i_service_req.request_cmd = TO_BOOL(E_Util_Service_Req.On)  THEN 
		IF  (service_req_queue[idx_queue].rs_number = i_service_req.rs_number)  THEN
			service_assign := FALSE;
			EXIT;
		ELSE
			service_assign := TRUE;
		END_IF
		service_release := FALSE; // added to reset the req cmd
	END_IF
END_FOR

FOR idx_queue := 1 TO rs_count DO
	IF i_service_req.request_cmd = TO_BOOL(E_Util_Service_Req.Off)  THEN 
		IF  (service_req_queue[idx_queue].rs_number = i_service_req.rs_number)  THEN
			service_release := TRUE;
			EXIT;
		ELSE
			service_release := FALSE;
		END_IF
		service_assign := FALSE;   // added to reset the req cmd
	END_IF
END_FOR


trig_service_assign(CLK := service_assign);
trig_service_release(CLK := service_release);


IF trig_service_assign.Q THEN
	FOR idx_queue := 1 TO rs_count DO
		IF i_rs_module_constrain THEN
			IF idx_queue = i_shared_rs THEN 
				rs_same_module := Check_RSs_SameModule(i_rs_1 := service_req_queue[idx_queue-1].rs_number, i_rs_2 := i_service_req.rs_number);
			ELSE
				rs_same_module := Check_RSs_SameModule(i_rs_1 := service_req_queue[idx_queue].rs_number, i_rs_2 := i_service_req.rs_number);
			END_IF
		END_IF
		IF service_req_queue[idx_queue].rs_number = i_service_req.rs_number THEN
			EXIT;
		ELSIF NOT service_req_queue[idx_queue].is_assigned AND  (service_req_queue[idx_queue].rs_number <> i_service_req.rs_number)  THEN 
				IF i_rs_module_constrain AND  (idx_queue = i_shared_rs) AND  rs_same_module THEN 
					CONTINUE;
				ELSE
					service_req_queue[idx_queue].is_assigned  := TRUE;
					service_req_queue[idx_queue].rs_number := i_service_req.rs_number;
					o_passiveQueue_number[idx_queue]		:= service_req_queue[idx_queue].rs_number;
					EXIT;
				END_IF
		END_IF
	END_FOR
END_IF



// Remove from queue
IF trig_service_release.Q THEN
	FOR idx_queue := 1 TO rs_count DO
		IF service_req_queue[idx_queue].rs_number =  i_service_req.rs_number THEN
			service_req_queue[idx_queue].rs_number := 0;
			service_req_queue[idx_queue].is_assigned  := FALSE;
			o_passiveQueue_number[idx_queue] 	:= service_req_queue[idx_queue].rs_number;
			EXIT;
		END_IF
	END_FOR
END_IF

// Update queue

FOR idx_queue := 1 TO rs_count DO
	IF  NOT service_req_queue[idx_queue].is_assigned  THEN 
		FOR idx_queue_update := idx_queue + 1 TO rs_count DO
			IF i_rs_module_constrain THEN
				IF idx_queue = i_shared_rs THEN 
					rs_same_module := Check_RSs_SameModule(i_rs_1 := service_req_queue[idx_queue-1].rs_number, i_rs_2 := service_req_queue[idx_queue_update].rs_number);
				ELSE
					rs_same_module := Check_RSs_SameModule(i_rs_1 := service_req_queue[idx_queue].rs_number, i_rs_2 := service_req_queue[idx_queue_update].rs_number);
				END_IF
			END_IF
			IF service_req_queue[idx_queue_update].rs_number > 0 THEN 
				IF  NOT i_rs_module_constrain THEN 
					service_req_queue[idx_queue] := service_req_queue[idx_queue_update];
					service_req_queue[idx_queue_update].rs_number := 0;
					service_req_queue[idx_queue_update].is_assigned := FALSE;
					o_passiveQueue_number[idx_queue]:=service_req_queue[idx_queue].rs_number;
					o_passiveQueue_number[idx_queue_update] := 0;
					EXIT;
				ELSIF i_rs_module_constrain AND NOT (idx_queue = i_shared_rs) THEN 
					service_req_queue[idx_queue] := service_req_queue[idx_queue_update];
					service_req_queue[idx_queue_update].rs_number := 0;
					service_req_queue[idx_queue_update].is_assigned := FALSE;
					o_passiveQueue_number[idx_queue]:=service_req_queue[idx_queue].rs_number;
					o_passiveQueue_number[idx_queue_update] := 0;
					EXIT;
				ELSIF i_rs_module_constrain AND  (idx_queue = i_shared_rs) AND NOT rs_same_module THEN
					service_req_queue[idx_queue] := service_req_queue[idx_queue_update];
					service_req_queue[idx_queue_update].rs_number := 0;
					service_req_queue[idx_queue_update].is_assigned := FALSE;
					o_passiveQueue_number[idx_queue]:=service_req_queue[idx_queue].rs_number;
					o_passiveQueue_number[idx_queue_update] := 0;
					EXIT;
				ELSIF i_rs_module_constrain AND  (idx_queue = i_shared_rs) AND  rs_same_module THEN
					CONTINUE;				
				END_IF
			END_IF						
		END_FOR	
	END_IF
END_FOR

// Service on/off requet to Utilities

o_service_req := service_req_queue[1].is_assigned ; // on request to utilities if queue pos #1 is populated / has a RS assigned 


// Service assigned sts to RS controller

IF i_shared_rs >= 2 THEN
	FOR idx_queue := 1 TO i_shared_rs DO 
		IF service_req_queue[idx_queue].is_assigned THEN 
			o_assigned_rs_number[idx_queue] := service_req_queue[idx_queue].rs_number;
		ELSE
			o_assigned_rs_number[idx_queue] := 0;
		END_IF
	END_FOR
ELSIF i_shared_rs = 1 THEN
	IF service_req_queue[idx_queue].is_assigned THEN 
		o_assigned_rs_number[1] := service_req_queue[1].rs_number;
	ELSE
		o_assigned_rs_number[1] := 0;
	END_IF
END_IF

METHOD Check_RSs_SameModule : BOOL
VAR_INPUT
	i_rs_1 : UINT;
	i_rs_2 : UINT;
END_VAR

Check_RSs_SameModule := ((i_rs_1 >=1  AND i_rs_1 <= 3) AND (i_rs_2 >=1  AND i_rs_2 <= 3)) OR 
						((i_rs_1 >=4  AND i_rs_1 <= 6) AND (i_rs_2 >=4  AND i_rs_2 <= 6)) OR 
                        ((i_rs_1 >=7  AND i_rs_1 <= 9) AND (i_rs_2 >=7  AND i_rs_2 <= 9)) OR
						((i_rs_1 >=10 AND i_rs_1<= 12) AND (i_rs_2 >=10 AND i_rs_2 <= 12));
END_METHOD

METHOD Clear_Queue : BOOL
VAR_INPUT
END_VAR
FOR idx_queue := 1 TO rs_count DO
	service_req_queue[idx_queue].rs_number := 0;
	service_req_queue[idx_queue].is_assigned  := FALSE;
	o_passiveQueue_number[idx_queue] 	:= service_req_queue[idx_queue].rs_number;
END_FOR
END_METHOD

END_FUNCTION_BLOCK

// ---- POUs/Reactor_Set_02/P_M01_RS02.TcPOU
PROGRAM P_M01_RS02
VAR_INPUT
	stop_rs_automode													: BOOL;
	clear_rs_pause												: BOOL;
	close_valves														: BOOL;
	close_all_doors														: BOOL;
	open_all_doors														: BOOL;
	retract_all_clamps													: BOOL;
	extend_all_clamps													: BOOL;
	open_repres_valves													: BOOL;
	close_repres_valves													: BOOL;
	co2_sensors_off														: BOOL;
	co2_inside_sensors_on												: BOOL;
	co2_outside_sensors_on												: BOOL;
	fan_vfd_percent														: REAL		:= 0;
END_VAR
VAR_OUTPUT
	repres_valves_clear													: BOOL;
	average_pressure_within_ambient										: BOOL;
	reactor_done														: BOOL;
	utility_error														: BOOL;
	cancel_reactor_set													: BOOL;
	cancel_all_reactor_sets												: BOOL;
	inlet_air_high_temp_count											: INT;
	open_inlet_doors													: BOOL;
	open_outlet_doors													: BOOL;
	close_inlet_doors													: BOOL;
	close_outlet_doors													: BOOL;
	open_doors															: BOOL;
	close_doors															: BOOL;
	inlet_door_clamps_extend											: BOOL;
	outlet_door_clamps_extend											: BOOL;
	inlet_door_clamps_retract											: BOOL;
	outlet_door_clamps_retract											: BOOL;
	extend_clamps														: BOOL;
	retract_clamps														: BOOL;
END_VAR
VAR
	R_S																	: Reactor_Set;

	fb_RS																: FB_Reactor_Set();
	fb_RS_IO															: FB_Reactor_Set_IO();
	fb_R1_IO															: FB_Reactor_IO();
	fb_R2_IO															: FB_Reactor_IO();
	fb_R3_IO															: FB_Reactor_IO();
	fb_R4_IO															: FB_Reactor_IO();
	
	fb_Fan_Vfd															: FB_Analog_Out();
	
	rAveragePressure													: REAL;
	rValve																: REAL;
	rPos																: REAL;
	rFanOldVfdPercent													: REAL		:= 0;
	
	iCount																: INT;
	iVacuumStatus														: INT;
	iError																: INT;
	
	bR1OverMaxPressure													: BOOL;
	bR2OverMaxPressure													: BOOL;
	bR3OverMaxPressure													: BOOL;
	bR4OverMaxPressure													: BOOL;
	
	bR1InletCO2Error													: BOOL;
	bR1InletH2OError													: BOOL;
	bR1OutletCO2Error													: BOOL;
	bR1OutletH2OError													: BOOL;
	bR1AirFlowError														: BOOL;
	bR1FilterDiffPresError												: BOOL;
	bR1SorbentDiffPresError												: BOOL;
	bR1FanDiffPresError													: BOOL;
	bR1ReactorPresError													: BOOL;
	
	bR2InletCO2Error													: BOOL;
	bR2InletH2OError													: BOOL;
	bR2OutletCO2Error													: BOOL;
	bR2OutletH2OError													: BOOL;
	bR2AirFlowError														: BOOL;
	bR2FilterDiffPresError												: BOOL;
	bR2SorbentDiffPresError												: BOOL;
	bR2FanDiffPresError													: BOOL;
	bR2ReactorPresError													: BOOL;
	
	bR3InletCO2Error													: BOOL;
	bR3InletH2OError													: BOOL;
	bR3OutletCO2Error													: BOOL;
	bR3OutletH2OError													: BOOL;
	bR3AirFlowError														: BOOL;
	bR3FilterDiffPresError												: BOOL;
	bR3SorbentDiffPresError												: BOOL;
	bR3FanDiffPresError													: BOOL;
	bR3ReactorPresError													: BOOL;
	
	bR4InletCO2Error													: BOOL;
	bR4InletH2OError													: BOOL;
	bR4OutletCO2Error													: BOOL;
	bR4OutletH2OError													: BOOL;
	bR4AirFlowError														: BOOL;
	bR4FilterDiffPresError												: BOOL;
	bR4SorbentDiffPresError												: BOOL;
	bR4FanDiffPresError													: BOOL;
	bR4ReactorPresError													: BOOL;
	
	stop_reactor_set													: BOOL;
	clear_reactor_set_pause												: BOOL;
END_VAR

// Phase 0 - P_M01_RS02
// Rev 1.0 - May 11, 2024

giEvacuationErrorRS														:= SEL(giEvacuationErrorRS = 2, giEvacuationErrorRS, 0);
giDesorptionErrorRS														:= SEL(giDesorptionErrorRS = 2, giDesorptionErrorRS, 0);
giSafeShutdown1RS														:= SEL(giSafeShutdown1RS = 2, giSafeShutdown1RS, 0);
giSafeShutdown23RS														:= SEL(giSafeShutdown23RS = 2, giSafeShutdown23RS, 0);

stop_reactor_set														:= stop_rs_automode;
stop_rs_automode														:= FALSE;
clear_reactor_set_pause													:= clear_rs_pause;
clear_rs_pause															:= FALSE;

A_Reactor_Set();

// REACTOR OUTPUTS
IF open_repres_valves OR R_S.open_repres_valves THEN
	fb_R1_IO.bRepresValve												:= TRUE;
	fb_R2_IO.bRepresValve												:= TRUE;
	fb_R3_IO.bRepresValve												:= TRUE;
	fb_R4_IO.bRepresValve												:= TRUE;
	open_repres_valves													:= FALSE;
END_IF
IF close_repres_valves OR R_S.close_repres_valves THEN
	fb_R1_IO.bRepresValve												:= FALSE;
	fb_R2_IO.bRepresValve												:= FALSE;
	fb_R3_IO.bRepresValve												:= FALSE;
	fb_R4_IO.bRepresValve												:= FALSE;
	close_repres_valves													:= FALSE;
END_IF

repres_valves_clear														:= fb_R1_IO.repres_valve_clear AND fb_R2_IO.repres_valve_clear AND fb_R3_IO.repres_valve_clear AND fb_R4_IO.repres_valve_clear;
IF NOT repres_valves_clear THEN
	R_S.repres_valve_error												:= SEL(fb_R4_IO.repres_valve_clear, CONCAT(_R4, gsRepressurizationValveError), '');
	R_S.repres_valve_error												:= SEL(fb_R3_IO.repres_valve_clear, CONCAT(_R3, gsRepressurizationValveError), R_S.repres_valve_error);
	R_S.repres_valve_error												:= SEL(fb_R2_IO.repres_valve_clear, CONCAT(_R2, gsRepressurizationValveError), R_S.repres_valve_error);
	R_S.repres_valve_error												:= SEL(fb_R1_IO.repres_valve_clear, CONCAT(_R1, gsRepressurizationValveError), R_S.repres_valve_error);
ELSE
	R_S.repres_valve_error												:= '';
END_IF

fb_Fan_Vfd(Input1:= fan_vfd_percent, Input2:= R_S.fan_vfd_percent);
IF fan_vfd_percent <> rFanOldVfdPercent THEN
	fb_R1_IO.fan_vfd_input											:= fan_vfd_percent;
	fb_R2_IO.fan_vfd_input											:= fan_vfd_percent;
	fb_R3_IO.fan_vfd_input											:= fan_vfd_percent;
	fb_R4_IO.fan_vfd_input											:= fan_vfd_percent;
	rFanOldVfdPercent													:= fan_vfd_percent;
END_IF
		
A_Reactor1_IO();
A_Reactor2_IO();
A_Reactor3_IO();
A_Reactor4_IO();

inlet_air_high_temp_count												:= fb_R1_IO.adsorption_high_temp_count + fb_R2_IO.adsorption_high_temp_count + fb_R3_IO.adsorption_high_temp_count + fb_R4_IO.adsorption_high_temp_count;
R_S.inlet_air_high_temp_count											:= inlet_air_high_temp_count;
R_S.desorption_high_temp_count											:= fb_R1_IO.desorption_high_temp_count + fb_R2_IO.desorption_high_temp_count + fb_R3_IO.desorption_high_temp_count + fb_R4_IO.desorption_high_temp_count;
R_S.vacuum_cooling_high_temp_count										:= fb_R1_IO.vacuum_cooling_high_temp_count + fb_R2_IO.vacuum_cooling_high_temp_count + fb_R3_IO.vacuum_cooling_high_temp_count + fb_R4_IO.vacuum_cooling_high_temp_count;
R_S.sorbent_high_temp													:= F_HighestReal(fb_R1_IO.sorbent_high_temp, fb_R2_IO.sorbent_high_temp, fb_R3_IO.sorbent_high_temp, fb_R4_IO.sorbent_high_temp);

m01_rs2_r1.reactor_wall_temp											:= F_Temperature(m01_rs2_r1.TT_05, m01_rs2_r1.reactor_wall_temp_offset);
m01_rs2_r1.outlet_line_temp												:= F_Temperature(m01_rs2_r1.TT_06, m01_rs2_r1.outlet_line_temp_offset);
m01_rs2_r2.reactor_wall_temp											:= F_Temperature(m01_rs2_r2.TT_05, m01_rs2_r2.reactor_wall_temp_offset);
m01_rs2_r2.outlet_line_temp												:= F_Temperature(m01_rs2_r2.TT_06, m01_rs2_r2.outlet_line_temp_offset);
m01_rs2_r3.reactor_wall_temp											:= F_Temperature(m01_rs2_r3.TT_05, m01_rs2_r3.reactor_wall_temp_offset);
m01_rs2_r3.outlet_line_temp												:= F_Temperature(m01_rs2_r3.TT_06, m01_rs2_r3.outlet_line_temp_offset);
m01_rs2_r4.reactor_wall_temp											:= F_Temperature(m01_rs2_r4.TT_05, m01_rs2_r4.reactor_wall_temp_offset);
m01_rs2_r4.outlet_line_temp												:= F_Temperature(m01_rs2_r4.TT_06, m01_rs2_r4.outlet_line_temp_offset);

// CO2 SENSOR HANDLING
IF co2_sensors_off OR R_S.co2_sensors_off THEN
	fb_R1_IO.co2_sensor_config											:= 0;
	fb_R2_IO.co2_sensor_config											:= 0;
	fb_R3_IO.co2_sensor_config											:= 0;
	fb_R4_IO.co2_sensor_config											:= 0;
	co2_sensors_off														:= FALSE;
ELSIF co2_inside_sensors_on OR R_S.co2_inside_sensors_on THEN
	fb_R1_IO.co2_sensor_config											:= 1;
	fb_R2_IO.co2_sensor_config											:= 1;
	fb_R3_IO.co2_sensor_config											:= 1;
	fb_R4_IO.co2_sensor_config											:= 1;
	co2_inside_sensors_on												:= FALSE;
ELSIF co2_outside_sensors_on OR R_S.co2_outside_sensors_on THEN
	fb_R1_IO.co2_sensor_config											:= 2;
	fb_R2_IO.co2_sensor_config											:= 2;
	fb_R3_IO.co2_sensor_config											:= 2;
	fb_R4_IO.co2_sensor_config											:= 2;
	co2_outside_sensors_on												:= FALSE;
END_IF
 
// DOORS & CLAMPS
inlet_door_clamps_extend												:= FALSE;	
outlet_door_clamps_extend												:= FALSE;
inlet_door_clamps_retract												:= FALSE;	
outlet_door_clamps_retract												:= FALSE;
extend_clamps															:= FALSE;
retract_clamps															:= FALSE;
IF extend_all_clamps OR R_S.extend_all_clamps THEN
	extend_clamps														:= TRUE;
	extend_all_clamps													:= FALSE;
END_IF
IF retract_all_clamps OR R_S.retract_all_clamps THEN
	retract_clamps														:= TRUE;	
	retract_all_clamps													:= FALSE;
END_IF
R_S.all_clamps_extended													:= fb_R1_IO.door_clamps_extended AND fb_R2_IO.door_clamps_extended AND fb_R3_IO.door_clamps_extended AND fb_R4_IO.door_clamps_extended; 
R_S.all_clamps_retracted												:= fb_R1_IO.door_clamps_retracted AND fb_R2_IO.door_clamps_retracted AND fb_R3_IO.door_clamps_retracted AND fb_R4_IO.door_clamps_retracted;

open_inlet_doors														:= FALSE;
open_outlet_doors														:= FALSE;
close_inlet_doors														:= FALSE;
close_outlet_doors														:= FALSE;
open_doors																:= FALSE;
close_doors																:= FALSE;
IF open_all_doors OR R_S.open_all_doors THEN
	open_doors															:= TRUE;
	open_all_doors														:= FALSE;
END_IF
fb_R1_IO.close_doors													:= FALSE;
IF close_all_doors OR R_S.close_all_doors THEN
	close_doors															:= TRUE;
	close_all_doors														:= FALSE;
END_IF
R_S.all_doors_open														:= fb_R1_IO.doors_open AND fb_R2_IO.doors_open AND fb_R3_IO.doors_open AND fb_R4_IO.doors_open;
R_S.all_doors_closed													:= fb_R1_IO.doors_closed AND fb_R2_IO.doors_closed AND fb_R3_IO.doors_closed AND fb_R4_IO.doors_closed;

m01_rs2_r1.inlet_co2													:= F_AnalogIn(m01_rs2_r1.AT_01, m01_rs2_r1.inlet_co2_low, m01_rs2_r1.inlet_co2_high, m01_rs2_r1.inlet_co2_min, m01_rs2_r1.inlet_co2_offset);
bR1InletCO2Error														:= P_Alarms.M_Check_Error(m01_rs2_r1.inlet_co2_error, bR1InletCO2Error, CONCAT(_RS01, _R1), gsInletCO2SensorError, gsProcessWillContinue);
m01_rs2_r1.inlet_h2o													:= F_AnalogIn(m01_rs2_r1.AT_02, m01_rs2_r1.inlet_h2o_low, m01_rs2_r1.inlet_h2o_high, m01_rs2_r1.inlet_h2o_min, m01_rs2_r1.inlet_h2o_offset);
bR1InletH2OError														:= P_Alarms.M_Check_Error(m01_rs2_r1.inlet_h2o_error, bR1InletH2OError, CONCAT(_RS01, _R1), gsInletH2OSensorError, gsProcessWillContinue);
m01_rs2_r1.outlet_co2													:= F_AnalogIn(m01_rs2_r1.AT_03, m01_rs2_r1.outlet_co2_low, m01_rs2_r1.outlet_co2_high, m01_rs2_r1.outlet_co2_min, m01_rs2_r1.outlet_co2_offset);
bR1OutletCO2Error														:= P_Alarms.M_Check_Error(m01_rs2_r1.outlet_co2_error, bR1OutletCO2Error, CONCAT(_RS01, _R1), gsOutletCO2SensorError, gsProcessWillContinue);
m01_rs2_r1.outlet_h2o													:= F_AnalogIn(m01_rs2_r1.AT_04, m01_rs2_r1.outlet_h2o_low, m01_rs2_r1.outlet_h2o_high, m01_rs2_r1.outlet_h2o_min, m01_rs2_r1.outlet_h2o_offset);
bR1OutletH2OError														:= P_Alarms.M_Check_Error(m01_rs2_r1.outlet_h2o_error, bR1OutletH2OError, CONCAT(_RS01, _R1), gsOutletH2OSensorError, gsProcessWillContinue);
m01_rs2_r1.air_flow														:= F_AnalogIn(m01_rs2_r1.FT_01, m01_rs2_r1.air_flow_low, m01_rs2_r1.air_flow_high, m01_rs2_r1.air_flow_min, m01_rs2_r1.air_flow_offset);
bR1AirFlowError															:= P_Alarms.M_Check_Error(m01_rs2_r1.air_flow_error, bR1AirFlowError, CONCAT(_RS01, _R1), gsAirFlowSensorError, gsProcessWillContinue);
m01_rs2_r1.filter_diff_pres												:= F_AnalogIn(m01_rs2_r1.PDT_01, m01_rs2_r1.filter_diff_pres_low, m01_rs2_r1.filter_diff_pres_high, m01_rs2_r1.filter_diff_pres_min, m01_rs2_r1.filter_diff_pres_offset);
bR1FilterDiffPresError													:= P_Alarms.M_Check_Error(m01_rs2_r1.filter_diff_pres_error, bR1FilterDiffPresError, CONCAT(_RS01, _R1), gsFilterDiffPresSensorError, gsProcessWillContinue);
m01_rs2_r1.sorbent_diff_pres											:= F_AnalogIn(m01_rs2_r1.PDT_02, m01_rs2_r1.sorbent_diff_pres_low, m01_rs2_r1.sorbent_diff_pres_high, m01_rs2_r1.sorbent_diff_pres_min, m01_rs2_r1.sorbent_diff_pres_offset,);
bR1SorbentDiffPresError													:= P_Alarms.M_Check_Error(m01_rs2_r1.sorbent_diff_pres_error, bR1SorbentDiffPresError, CONCAT(_RS01, _R1), gsSorbentDiffPresSensorError, gsProcessWillContinue);
m01_rs2_r1.fan_diff_pres												:= F_AnalogIn(m01_rs2_r1.PDT_03, m01_rs2_r1.fan_diff_pres_low, m01_rs2_r1.fan_diff_pres_high, m01_rs2_r1.fan_diff_pres_min, m01_rs2_r1.fan_diff_pres_offset);
bR1FanDiffPresError														:= P_Alarms.M_Check_Error(m01_rs2_r1.fan_diff_pres_error, bR1FanDiffPresError, CONCAT(_RS01, _R1), gsFanDiffPresSensorError, gsProcessWillContinue);
m01_rs2_r1.reactor_pres													:= F_AnalogIn(m01_rs2_r1.PT_01, m01_rs2_r1.reactor_pres_low, m01_rs2_r1.reactor_pres_high, m01_rs2_r1.reactor_pres_min, m01_rs2_r1.reactor_pres_offset);
bR1ReactorPresError														:= P_Alarms.M_Check_Error(m01_rs2_r1.reactor_pres_error, bR1ReactorPresError, CONCAT(_RS01, _R1), gsReactorPresSensorError, gsProcessWillContinue);
R_S.R1_reactor_pres														:= m01_rs2_r1.reactor_pres;
R_S.R1_reactor_pres_error												:= bR1ReactorPresError;
bR1OverMaxPressure														:= NOT m01_rs2_r1.reactor_pres_error AND m01_rs2_r1.reactor_pres > m01.SP_maximum_safe_reactor_steam_pressure;

m01_rs2_r2.inlet_co2													:= F_AnalogIn(m01_rs2_r2.AT_01, m01_rs2_r2.inlet_co2_low, m01_rs2_r2.inlet_co2_high, m01_rs2_r2.inlet_co2_min, m01_rs2_r2.inlet_co2_offset);
bR2InletCO2Error														:= P_Alarms.M_Check_Error(m01_rs2_r2.inlet_co2_error, bR2InletCO2Error, CONCAT(_RS01, _R2), gsInletCO2SensorError, gsProcessWillContinue);
m01_rs2_r2.inlet_h2o													:= F_AnalogIn(m01_rs2_r2.AT_02, m01_rs2_r2.inlet_h2o_low, m01_rs2_r2.inlet_h2o_high, m01_rs2_r2.inlet_h2o_min, m01_rs2_r2.inlet_h2o_offset);
bR2InletH2OError														:= P_Alarms.M_Check_Error(m01_rs2_r2.inlet_h2o_error, bR2InletH2OError, CONCAT(_RS01, _R2), gsInletH2OSensorError, gsProcessWillContinue);
m01_rs2_r2.outlet_co2													:= F_AnalogIn(m01_rs2_r2.AT_03, m01_rs2_r2.outlet_co2_low, m01_rs2_r2.outlet_co2_high, m01_rs2_r2.outlet_co2_min, m01_rs2_r2.outlet_co2_offset);
bR2OutletCO2Error														:= P_Alarms.M_Check_Error(m01_rs2_r2.outlet_co2_error, bR2OutletCO2Error, CONCAT(_RS01, _R2), gsOutletCO2SensorError, gsProcessWillContinue);
m01_rs2_r2.outlet_h2o													:= F_AnalogIn(m01_rs2_r2.AT_04, m01_rs2_r2.outlet_h2o_low, m01_rs2_r2.outlet_h2o_high, m01_rs2_r2.outlet_h2o_min, m01_rs2_r2.outlet_h2o_offset);
bR2OutletH2OError														:= P_Alarms.M_Check_Error(m01_rs2_r2.outlet_h2o_error, bR2OutletH2OError, CONCAT(_RS01, _R2), gsOutletH2OSensorError, gsProcessWillContinue);
m01_rs2_r2.air_flow														:= F_AnalogIn(m01_rs2_r2.FT_01, m01_rs2_r2.air_flow_low, m01_rs2_r2.air_flow_high, m01_rs2_r2.air_flow_min, m01_rs2_r2.air_flow_offset);
bR2AirFlowError															:= P_Alarms.M_Check_Error(m01_rs2_r2.air_flow_error, bR2AirFlowError, CONCAT(_RS01, _R2), gsAirFlowSensorError, gsProcessWillContinue);
m01_rs2_r2.filter_diff_pres												:= F_AnalogIn(m01_rs2_r2.PDT_01, m01_rs2_r2.filter_diff_pres_low, m01_rs2_r2.filter_diff_pres_high, m01_rs2_r2.filter_diff_pres_min, m01_rs2_r2.filter_diff_pres_offset);
bR2FilterDiffPresError													:= P_Alarms.M_Check_Error(m01_rs2_r2.filter_diff_pres_error, bR2FilterDiffPresError, CONCAT(_RS01, _R2), gsFilterDiffPresSensorError, gsProcessWillContinue);
m01_rs2_r2.sorbent_diff_pres											:= F_AnalogIn(m01_rs2_r2.PDT_02, m01_rs2_r2.sorbent_diff_pres_low, m01_rs2_r2.sorbent_diff_pres_high, m01_rs2_r2.sorbent_diff_pres_min, m01_rs2_r2.sorbent_diff_pres_offset,);
bR2SorbentDiffPresError													:= P_Alarms.M_Check_Error(m01_rs2_r2.sorbent_diff_pres_error, bR2SorbentDiffPresError, CONCAT(_RS01, _R2), gsSorbentDiffPresSensorError, gsProcessWillContinue);
m01_rs2_r2.fan_diff_pres												:= F_AnalogIn(m01_rs2_r2.PDT_03, m01_rs2_r2.fan_diff_pres_low, m01_rs2_r2.fan_diff_pres_high, m01_rs2_r2.fan_diff_pres_min, m01_rs2_r2.fan_diff_pres_offset);
bR2FanDiffPresError														:= P_Alarms.M_Check_Error(m01_rs2_r2.fan_diff_pres_error, bR2FanDiffPresError, CONCAT(_RS01, _R2), gsFanDiffPresSensorError, gsProcessWillContinue);
m01_rs2_r2.reactor_pres													:= F_AnalogIn(m01_rs2_r2.PT_01, m01_rs2_r2.reactor_pres_low, m01_rs2_r2.reactor_pres_high, m01_rs2_r2.reactor_pres_min, m01_rs2_r2.reactor_pres_offset);
bR2ReactorPresError														:= P_Alarms.M_Check_Error(m01_rs2_r2.reactor_pres_error, bR2ReactorPresError, CONCAT(_RS01, _R2), gsReactorPresSensorError, gsProcessWillContinue);
R_S.R2_reactor_pres														:= m01_rs2_r2.reactor_pres;
R_S.R2_reactor_pres_error												:= bR2ReactorPresError;
bR2OverMaxPressure														:= NOT m01_rs2_r2.reactor_pres_error AND m01_rs2_r2.reactor_pres > m01.SP_maximum_safe_reactor_steam_pressure;

m01_rs2_r3.inlet_co2													:= F_AnalogIn(m01_rs2_r3.AT_01, m01_rs2_r3.inlet_co2_low, m01_rs2_r3.inlet_co2_high, m01_rs2_r3.inlet_co2_min, m01_rs2_r3.inlet_co2_offset);
bR3InletCO2Error														:= P_Alarms.M_Check_Error(m01_rs2_r3.inlet_co2_error, bR3InletCO2Error, CONCAT(_RS01, _R3), gsInletCO2SensorError, gsProcessWillContinue);
m01_rs2_r3.inlet_h2o													:= F_AnalogIn(m01_rs2_r3.AT_02, m01_rs2_r3.inlet_h2o_low, m01_rs2_r3.inlet_h2o_high, m01_rs2_r3.inlet_h2o_min, m01_rs2_r3.inlet_h2o_offset);
bR3InletH2OError														:= P_Alarms.M_Check_Error(m01_rs2_r3.inlet_h2o_error, bR3InletH2OError, CONCAT(_RS01, _R3), gsInletH2OSensorError, gsProcessWillContinue);
m01_rs2_r3.outlet_co2													:= F_AnalogIn(m01_rs2_r3.AT_03, m01_rs2_r3.outlet_co2_low, m01_rs2_r3.outlet_co2_high, m01_rs2_r3.outlet_co2_min, m01_rs2_r3.outlet_co2_offset);
bR3OutletCO2Error														:= P_Alarms.M_Check_Error(m01_rs2_r3.outlet_co2_error, bR3OutletCO2Error, CONCAT(_RS01, _R3), gsOutletCO2SensorError, gsProcessWillContinue);
m01_rs2_r3.outlet_h2o													:= F_AnalogIn(m01_rs2_r3.AT_04, m01_rs2_r3.outlet_h2o_low, m01_rs2_r3.outlet_h2o_high, m01_rs2_r3.outlet_h2o_min, m01_rs2_r3.outlet_h2o_offset);
bR3OutletH2OError														:= P_Alarms.M_Check_Error(m01_rs2_r3.outlet_h2o_error, bR3OutletH2OError, CONCAT(_RS01, _R3), gsOutletH2OSensorError, gsProcessWillContinue);
m01_rs2_r3.air_flow														:= F_AnalogIn(m01_rs2_r3.FT_01, m01_rs2_r3.air_flow_low, m01_rs2_r3.air_flow_high, m01_rs2_r3.air_flow_min, m01_rs2_r3.air_flow_offset);
bR3AirFlowError															:= P_Alarms.M_Check_Error(m01_rs2_r3.air_flow_error, bR3AirFlowError, CONCAT(_RS01, _R3), gsAirFlowSensorError, gsProcessWillContinue);
m01_rs2_r3.filter_diff_pres												:= F_AnalogIn(m01_rs2_r3.PDT_01, m01_rs2_r3.filter_diff_pres_low, m01_rs2_r3.filter_diff_pres_high, m01_rs2_r3.filter_diff_pres_min, m01_rs2_r3.filter_diff_pres_offset);
bR3FilterDiffPresError													:= P_Alarms.M_Check_Error(m01_rs2_r3.filter_diff_pres_error, bR3FilterDiffPresError, CONCAT(_RS01, _R3), gsFilterDiffPresSensorError, gsProcessWillContinue);
m01_rs2_r3.sorbent_diff_pres											:= F_AnalogIn(m01_rs2_r3.PDT_02, m01_rs2_r3.sorbent_diff_pres_low, m01_rs2_r3.sorbent_diff_pres_high, m01_rs2_r3.sorbent_diff_pres_min, m01_rs2_r3.sorbent_diff_pres_offset,);
bR3SorbentDiffPresError													:= P_Alarms.M_Check_Error(m01_rs2_r3.sorbent_diff_pres_error, bR3SorbentDiffPresError, CONCAT(_RS01, _R3), gsSorbentDiffPresSensorError, gsProcessWillContinue);
m01_rs2_r3.fan_diff_pres												:= F_AnalogIn(m01_rs2_r3.PDT_03, m01_rs2_r3.fan_diff_pres_low, m01_rs2_r3.fan_diff_pres_high, m01_rs2_r3.fan_diff_pres_min, m01_rs2_r3.fan_diff_pres_offset);
bR3FanDiffPresError														:= P_Alarms.M_Check_Error(m01_rs2_r3.fan_diff_pres_error, bR3FanDiffPresError, CONCAT(_RS01, _R3), gsFanDiffPresSensorError, gsProcessWillContinue);
m01_rs2_r3.reactor_pres													:= F_AnalogIn(m01_rs2_r3.PT_01, m01_rs2_r3.reactor_pres_low, m01_rs2_r3.reactor_pres_high, m01_rs2_r3.reactor_pres_min, m01_rs2_r3.reactor_pres_offset);
bR3ReactorPresError														:= P_Alarms.M_Check_Error(m01_rs2_r3.reactor_pres_error, bR3ReactorPresError, CONCAT(_RS01, _R3), gsReactorPresSensorError, gsProcessWillContinue);
R_S.R3_reactor_pres														:= m01_rs2_r3.reactor_pres;
R_S.R3_reactor_pres_error												:= bR3ReactorPresError;
bR3OverMaxPressure														:= NOT m01_rs2_r3.reactor_pres_error AND m01_rs2_r3.reactor_pres > m01.SP_maximum_safe_reactor_steam_pressure;

m01_rs2_r4.inlet_co2													:= F_AnalogIn(m01_rs2_r4.AT_01, m01_rs2_r4.inlet_co2_low, m01_rs2_r4.inlet_co2_high, m01_rs2_r4.inlet_co2_min, m01_rs2_r4.inlet_co2_offset);
bR4InletCO2Error														:= P_Alarms.M_Check_Error(m01_rs2_r4.inlet_co2_error, bR4InletCO2Error, CONCAT(_RS01, _R4), gsInletCO2SensorError, gsProcessWillContinue);
m01_rs2_r4.inlet_h2o													:= F_AnalogIn(m01_rs2_r4.AT_02, m01_rs2_r4.inlet_h2o_low, m01_rs2_r4.inlet_h2o_high, m01_rs2_r4.inlet_h2o_min, m01_rs2_r4.inlet_h2o_offset);
bR4InletH2OError														:= P_Alarms.M_Check_Error(m01_rs2_r4.inlet_h2o_error, bR4InletH2OError, CONCAT(_RS01, _R4), gsInletH2OSensorError, gsProcessWillContinue);
m01_rs2_r4.outlet_co2													:= F_AnalogIn(m01_rs2_r4.AT_03, m01_rs2_r4.outlet_co2_low, m01_rs2_r4.outlet_co2_high, m01_rs2_r4.outlet_co2_min, m01_rs2_r4.outlet_co2_offset);
bR4OutletCO2Error														:= P_Alarms.M_Check_Error(m01_rs2_r4.outlet_co2_error, bR4OutletCO2Error, CONCAT(_RS01, _R4), gsOutletCO2SensorError, gsProcessWillContinue);
m01_rs2_r4.outlet_h2o													:= F_AnalogIn(m01_rs2_r4.AT_04, m01_rs2_r4.outlet_h2o_low, m01_rs2_r4.outlet_h2o_high, m01_rs2_r4.outlet_h2o_min, m01_rs2_r4.outlet_h2o_offset);
bR4OutletH2OError														:= P_Alarms.M_Check_Error(m01_rs2_r4.outlet_h2o_error, bR4OutletH2OError, CONCAT(_RS01, _R4), gsOutletH2OSensorError, gsProcessWillContinue);
m01_rs2_r4.air_flow														:= F_AnalogIn(m01_rs2_r4.FT_01, m01_rs2_r4.air_flow_low, m01_rs2_r4.air_flow_high, m01_rs2_r4.air_flow_min, m01_rs2_r4.air_flow_offset);
bR4AirFlowError															:= P_Alarms.M_Check_Error(m01_rs2_r4.air_flow_error, bR4AirFlowError, CONCAT(_RS01, _R4), gsAirFlowSensorError, gsProcessWillContinue);
m01_rs2_r4.filter_diff_pres												:= F_AnalogIn(m01_rs2_r4.PDT_01, m01_rs2_r4.filter_diff_pres_low, m01_rs2_r4.filter_diff_pres_high, m01_rs2_r4.filter_diff_pres_min, m01_rs2_r4.filter_diff_pres_offset);
bR4FilterDiffPresError													:= P_Alarms.M_Check_Error(m01_rs2_r4.filter_diff_pres_error, bR4FilterDiffPresError, CONCAT(_RS01, _R4), gsFilterDiffPresSensorError, gsProcessWillContinue);
m01_rs2_r4.sorbent_diff_pres											:= F_AnalogIn(m01_rs2_r4.PDT_02, m01_rs2_r4.sorbent_diff_pres_low, m01_rs2_r4.sorbent_diff_pres_high, m01_rs2_r4.sorbent_diff_pres_min, m01_rs2_r4.sorbent_diff_pres_offset,);
bR4SorbentDiffPresError													:= P_Alarms.M_Check_Error(m01_rs2_r4.sorbent_diff_pres_error, bR4SorbentDiffPresError, CONCAT(_RS01, _R4), gsSorbentDiffPresSensorError, gsProcessWillContinue);
m01_rs2_r4.fan_diff_pres												:= F_AnalogIn(m01_rs2_r4.PDT_03, m01_rs2_r4.fan_diff_pres_low, m01_rs2_r4.fan_diff_pres_high, m01_rs2_r4.fan_diff_pres_min, m01_rs2_r4.fan_diff_pres_offset);
bR4FanDiffPresError														:= P_Alarms.M_Check_Error(m01_rs2_r4.fan_diff_pres_error, bR4FanDiffPresError, CONCAT(_RS01, _R4), gsFanDiffPresSensorError, gsProcessWillContinue);
m01_rs2_r4.reactor_pres													:= F_AnalogIn(m01_rs2_r4.PT_01, m01_rs2_r4.reactor_pres_low, m01_rs2_r4.reactor_pres_high, m01_rs2_r4.reactor_pres_min, m01_rs2_r4.reactor_pres_offset);
bR4ReactorPresError														:= P_Alarms.M_Check_Error(m01_rs2_r4.reactor_pres_error, bR4ReactorPresError, CONCAT(_RS01, _R4), gsReactorPresSensorError, gsProcessWillContinue);
R_S.R4_reactor_pres														:= m01_rs2_r4.reactor_pres;
R_S.R4_reactor_pres_error												:= bR4ReactorPresError;
bR4OverMaxPressure														:= NOT m01_rs2_r4.reactor_pres_error AND m01_rs2_r4.reactor_pres > m01.SP_maximum_safe_reactor_steam_pressure;

rAveragePressure														:= 0;
iCount																	:= 0;
iVacuumStatus															:= 0;
iError																	:= 4;
IF NOT m01_rs2_r1.reactor_pres_error THEN
	rAveragePressure													:= rAveragePressure + m01_rs2_r1.reactor_pres;
	iVacuumStatus														:= F_LowMidHigh(m01_rs2_r1.reactor_pres, m01.SP_target_desorption_starting_pressure, m01.SP_maximum_desorption_starting_pressure, iVacuumStatus);
	iCount																:= iCount + 1;
	iError																:= iError - 1;
END_IF
IF NOT m01_rs2_r2.reactor_pres_error THEN
	rAveragePressure													:= rAveragePressure + m01_rs2_r2.reactor_pres;
	iVacuumStatus														:= F_LowMidHigh(m01_rs2_r2.reactor_pres, m01.SP_target_desorption_starting_pressure, m01.SP_maximum_desorption_starting_pressure, iVacuumStatus);
	iCount																:= iCount + 1;
	iError																:= iError - 1;
END_IF
IF NOT m01_rs2_r3.reactor_pres_error THEN
	rAveragePressure													:= rAveragePressure + m01_rs2_r3.reactor_pres;
	iVacuumStatus														:= F_LowMidHigh(m01_rs2_r3.reactor_pres, m01.SP_target_desorption_starting_pressure, m01.SP_maximum_desorption_starting_pressure, iVacuumStatus);
	iCount																:= iCount + 1;
	iError																:= iError - 1;
END_IF
IF NOT m01_rs2_r4.reactor_pres_error THEN
	rAveragePressure													:= rAveragePressure + m01_rs2_r4.reactor_pres;
	iVacuumStatus														:= F_LowMidHigh(m01_rs2_r1.reactor_pres, m01.SP_target_desorption_starting_pressure, m01.SP_maximum_desorption_starting_pressure, iVacuumStatus);
	iCount																:= iCount + 1;
	iError																:= iError - 1;
END_IF

R_S.average_reactor_pressure											:= SEL(iCount > 0, 0, rAveragePressure / iCount);
R_S.reactor_pressure_error												:= SEL(iError >= _MAX_REACTOR_ERRORS, '', F_Concat3(INT_TO_STRING(iError), ' ', gsReactorPresError));
R_S.reactor_vacuum_status												:= iVacuumStatus;
average_pressure_within_ambient											:= rAveragePressure >= P_M01.rMinPressureSP AND rAveragePressure <= P_M01.rMaxPressureSP;
R_S.average_reactor_pressure_within_ambient								:= average_pressure_within_ambient;
fb_RS_IO.reactor_over_max_pressure										:= bR1OverMaxPressure OR bR2OverMaxPressure OR bR3OverMaxPressure OR bR4OverMaxPressure;

R_S.R1_inlet_co2														:= m01_rs2_r1.inlet_co2;

R_S.R1_outlet_co2														:= m01_rs2_r1.outlet_co2;

ACTION A_Reactor_Set:
// Phase 0 - P_M01_RS02.A_Reactor_Set
// Rev 1.0 - May 10, 2024

fb_RS(		U															:= P_U01.u,
			R_S															:= P_M01_RS02.R_S,
			Stop_Reactor_Set											:= stop_reactor_set,
			Clear_Reactor_Set_Pause										:= clear_reactor_set_pause,
			test_error													:= gbRS02TestError,									///@@@ Temporary for testing
			RS_Name														:= _RS02,
			RS_Number													:= 2,
			Cycle_Mode													:= P_M01.sCycleModeRS02,
			Fan_Setpoint												:= m01.SP_reactor_set_2_vfd_percent,
//			Evac_Service_Acked											:= P_M01.evac_service_acked,
			Evac_Service_Assigned										:= P_M01.evac_service_assigned[2],
			Steam_Service_Assigned										:= P_M01.steam_service_assigned[2],
			Cycle_Stage													=> gsM01RS02CycleStage,
			Remaining_Time												=> m01_rs2.tr_Remaining_Time,
			Current_Step												=> m01_rs2.ti_Current_Step,
			Machine_State												=> m01_rs2.ti_Machine_State,
			Status														=> m01_rs2.ti_Status,
			Process_Running												=> m01_rs2.tb_Process_Running,
			Repressurization_Running									=> m01_rs2.tb_Repressurization_Running,
			Adsorption_Running											=> m01_rs2.tb_Adsorption_Running,
			Evacuation_Running											=> m01_rs2.tb_Evacuation_Running,
			Desorption_Running											=> m01_rs2.tb_Desorption_Running,
			Process_Complete											=> m01_rs2.tb_Process_Complete,
			Utility_Error												=> utility_error,
			Stop_M01_RS													=> stop_rs_automode,
			Cancel_Reactor_Set											=> cancel_reactor_set,
			Cancel_All_Reactor_Sets										=> cancel_all_reactor_sets,
			Done														=> reactor_done);

fb_RS_IO(	power_control_in											:= m01_rs2.power_control,
			power_control_out											=> m01_rs2.power_control_status,
			PWR_01														=> m01_rs2.PWR_01,
			power_control_fdbk_no										:= m01_rs2.circuit_breaker_no_feedback,
			power_control_fdbk_nc										:= m01_rs2.circuit_breaker_nc_feedback,
			condensate_lsl_in											:= m01_rs2.condensate_lsl,
			condensate_lsh_in											:= m01_rs2.condensate_lsh,
			condensate_lsl_out											=> R_S.condensate_lsl,
			condensate_lsh_out											=> R_S.condensate_lsh,
			condensate_pump_hmi											:= m01_rs2.condensate_pump,
			condensate_pump_plc											:= R_S.condensate_pump,
			condensate_pump_cmd_status									=> m01_rs2.condensate_pump_cmd_status,
			P_01														=> m01_rs2.P_01,
			rs_close_valves												:= R_S.close_all_valves,
			dead_air_valve_hmi											:= m01_rs2.dead_air_valve,
			dead_air_valve_plc											:= R_S.dead_air_valve,
			dead_air_valve_open_cmd_status								=> m01_rs2.dead_air_valve_open_cmd_status,
			dead_air_valve_open											:= m01_rs2.dead_air_valve_open,
			dead_air_valve_closed										:= m01_rs2.dead_air_valve_closed,
			dead_air_valve_clear										=> R_S.dead_air_valve_clear,
			XV_04														=> m01_rs2.XV_04,
			purge_valve_hmi												:= m01_rs2.purge_valve,
			purge_valve_plc												:= R_S.purge_valve,
			purge_valve_open_cmd_status									=> m01_rs2.purge_valve_open_cmd_status,
			purge_valve_open											:= m01_rs2.purge_valve_open,
			purge_valve_closed											:= m01_rs2.purge_valve_closed,
			purge_valve_clear											=> R_S.purge_valve_clear,
			XV_05														=> m01_rs2.XV_05,
			cooling_valve_hmi											:= m01_rs2.cooling_valve,
			cooling_valve_plc											:= R_S.cooling_valve,
			cooling_valve_open_cmd_status								=> m01_rs2.cooling_valve_open_cmd_status,
			cooling_valve_open											:= m01_rs2.cooling_valve_open,
			cooling_valve_closed										:= m01_rs2.cooling_valve_closed,
			cooling_valve_clear											=> R_S.cooling_valve_clear,
			XV_06														=> m01_rs2.XV_06,
			steam_header_valve_hmi										:= m01_rs2.steam_header_valve,
			steam_header_valve_plc										:= R_S.steam_header_valve,
			steam_header_valve_open_cmd_status							=> m01_rs2.steam_header_valve_open_cmd_status,
			steam_header_valve_open										:= m01_rs2.steam_header_valve_open,
			steam_header_valve_closed									:= m01_rs2.steam_header_valve_closed,
			steam_header_valve_not_closed								=> R_S.steam_header_valve_not_closed,
			steam_header_valve_clear									=> R_S.steam_header_valve_clear,
			XV_07														=> m01_rs2.XV_07,
			steam_control_valve_hmi										:= m01_rs2.steam_control_valve,
			steam_control_valve_plc										:= R_S.steam_control_valve,
			steam_control_valve_mode_hmi								:= m01_rs2.steam_control_valve_mode,
			steam_control_valve_mode_plc								:= R_S.steam_control_valve_mode,
			steam_control_valve_current_mode							=> m01_rs2.steam_control_valve_current_mode,
			steam_control_valve_error									:= m01_rs2.steam_control_valve_position_error,
			steam_control_valve_position								=> R_S.steam_control_valve_position,
			steam_control_valve_closed									=> R_S.steam_control_valve_closed,			
			steam_control_valve_setpoint								:= R_S.steam_control_valve_setpoint,
			steam_control_valve_control_point							:= R_S.steam_control_valve_control_point,
			steam_control_valve_loop_time								:= m01_rs2.steam_control_valve_loop_time,
			steam_control_valve_kp										:= m01_rs2.steam_control_valve_kp,
			steam_control_valve_ki										:= m01_rs2.steam_control_valve_ki,
			steam_control_valve_iband									:= m01_rs2.steam_control_valve_iband,
			steam_control_valve_base									:= m01_rs2.steam_control_valve_base,
			steam_control_valve_base_adjust								:= m01_rs2.steam_control_valve_base_adjust,
			PCV_01														=> m01_rs2.PCV_01,
			status_in													:= m01_rs2.ti_Status,
			status_out													=> m01_rs2.ts_Status_Text,
			valves_clear												=> R_S.valves_clear);
END_ACTION

ACTION A_Reactor1_IO:
// Phase 0 - P_M01_RS02.A_Reactor1_IO
// Rev 1.0 - April 26, 2024

fb_R1_IO(	RSet														:= _RS02,
			React														:= _R1,
			
			Power_On													:= m01_rs2.power_control,
			                                                    
			sorbent_low_temp											=> m01_rs2_r1.temp_low,
			sorbent_high_temp											=> m01_rs2_r1.temp_high,
			sorbent_average_temp										=> m01_rs2_r1.temp_average,
			                                                    
			TT_01_01													:= m01_rs2_r1._01_TT_01,
			TT_01_01_offset												:= m01_rs2_r1.cart01_front_temp_offset,
			TT_01_01_error												:= m01_rs2_r1._01_TT_01_Error,
			TT_01_03													:= m01_rs2_r1._01_TT_03,               
			TT_01_03_offset												:= m01_rs2_r1.cart01_front_temp_offset,
			TT_01_03_error												:= m01_rs2_r1._01_TT_03_Error,         
			TT_02_01													:= m01_rs2_r1._02_TT_01,               
			TT_02_01_offset												:= m01_rs2_r1.cart02_front_temp_offset,
			TT_02_01_error												:= m01_rs2_r1._02_TT_01_Error,         
			TT_02_03													:= m01_rs2_r1._02_TT_03,               
			TT_02_03_offset												:= m01_rs2_r1.cart02_front_temp_offset,
			TT_02_03_error												:= m01_rs2_r1._02_TT_03_Error,         
			TT_03_01													:= m01_rs2_r1._03_TT_01,               
			TT_03_01_offset												:= m01_rs2_r1.cart03_front_temp_offset,
			TT_03_01_error												:= m01_rs2_r1._03_TT_01_Error,         
			TT_03_03													:= m01_rs2_r1._03_TT_03,               
			TT_03_03_offset												:= m01_rs2_r1.cart03_front_temp_offset,
			TT_03_03_error												:= m01_rs2_r1._03_TT_03_Error,         
			TT_04_01													:= m01_rs2_r1._04_TT_01,               
			TT_04_01_offset												:= m01_rs2_r1.cart04_front_temp_offset,
			TT_04_01_error												:= m01_rs2_r1._04_TT_01_Error,         
			TT_04_03													:= m01_rs2_r1._04_TT_03,               
			TT_04_03_offset												:= m01_rs2_r1.cart04_front_temp_offset,
			TT_04_03_error												:= m01_rs2_r1._04_TT_03_Error,         
			TT_05_01													:= m01_rs2_r1._05_TT_01,               
			TT_05_01_offset												:= m01_rs2_r1.cart05_front_temp_offset,
			TT_05_01_error												:= m01_rs2_r1._05_TT_01_Error,         
			TT_05_03													:= m01_rs2_r1._05_TT_03,               
			TT_05_03_offset												:= m01_rs2_r1.cart05_front_temp_offset,
			TT_05_03_error												:= m01_rs2_r1._05_TT_03_Error,         
			TT_06_01													:= m01_rs2_r1._06_TT_01,               
			TT_06_01_offset												:= m01_rs2_r1.cart06_front_temp_offset,
			TT_06_01_error												:= m01_rs2_r1._06_TT_01_Error,         
			TT_06_03													:= m01_rs2_r1._06_TT_03,               
			TT_06_03_offset												:= m01_rs2_r1.cart06_front_temp_offset,
			TT_06_03_error												:= m01_rs2_r1._06_TT_03_Error,         
			TT_07_01													:= m01_rs2_r1._07_TT_01,               
			TT_07_01_offset												:= m01_rs2_r1.cart07_front_temp_offset,
			TT_07_01_error												:= m01_rs2_r1._07_TT_01_Error,         
			TT_07_03													:= m01_rs2_r1._07_TT_03,               
			TT_07_03_offset												:= m01_rs2_r1.cart07_front_temp_offset,
			TT_07_03_error												:= m01_rs2_r1._07_TT_03_Error,         
			TT_08_01													:= m01_rs2_r1._08_TT_01,               
			TT_08_01_offset												:= m01_rs2_r1.cart08_front_temp_offset,
			TT_08_01_error												:= m01_rs2_r1._08_TT_01_Error,         
			TT_08_03													:= m01_rs2_r1._08_TT_03,               
			TT_08_03_offset												:= m01_rs2_r1.cart08_front_temp_offset,
			TT_08_03_error												:= m01_rs2_r1._08_TT_03_Error,         
			TT_09_01													:= m01_rs2_r1._09_TT_01,               
			TT_09_01_offset												:= m01_rs2_r1.cart09_front_temp_offset,
			TT_09_01_error												:= m01_rs2_r1._09_TT_01_Error,         
			TT_09_03													:= m01_rs2_r1._09_TT_03,               
			TT_09_03_offset												:= m01_rs2_r1.cart09_front_temp_offset,
			TT_09_03_error												:= m01_rs2_r1._09_TT_03_Error,         
			TT_10_01													:= m01_rs2_r1._10_TT_01,               
			TT_10_01_offset												:= m01_rs2_r1.cart10_front_temp_offset,
			TT_10_01_error												:= m01_rs2_r1._10_TT_01_Error,         
			TT_10_03													:= m01_rs2_r1._10_TT_03,               
			TT_10_03_offset												:= m01_rs2_r1.cart10_front_temp_offset,
			TT_10_03_error												:= m01_rs2_r1._10_TT_03_Error,         
			TT_11_01													:= m01_rs2_r1._11_TT_01,               
			TT_11_01_offset												:= m01_rs2_r1.cart11_front_temp_offset,
			TT_11_01_error												:= m01_rs2_r1._11_TT_01_Error,         
			TT_11_03													:= m01_rs2_r1._11_TT_03,               
			TT_11_03_offset												:= m01_rs2_r1.cart11_front_temp_offset,
			TT_11_03_error												:= m01_rs2_r1._11_TT_03_Error,         
			TT_12_01													:= m01_rs2_r1._12_TT_01,               
			TT_12_01_offset												:= m01_rs2_r1.cart12_front_temp_offset,
			TT_12_01_error												:= m01_rs2_r1._12_TT_01_Error,         
			TT_12_03													:= m01_rs2_r1._12_TT_03,               
			TT_12_03_offset												:= m01_rs2_r1.cart12_front_temp_offset,
			TT_12_03_error												:= m01_rs2_r1._12_TT_03_Error,         
		    
			cart01_front_temp											=> m01_rs2_r1.cart01_front_temp,						
			cart01_front_temp_error 									=> m01_rs2_r1.cart01_front_temp_error,
			cart01_back_temp											=> m01_rs2_r1.cart01_back_temp,
			cart01_back_temp_error 										=> m01_rs2_r1.cart01_back_temp_error,
			cart02_front_temp											=> m01_rs2_r1.cart02_front_temp,						
			cart02_front_temp_error 									=> m01_rs2_r1.cart02_front_temp_error,
			cart02_back_temp											=> m01_rs2_r1.cart02_back_temp,
			cart02_back_temp_error 										=> m01_rs2_r1.cart02_back_temp_error,
			cart03_front_temp											=> m01_rs2_r1.cart03_front_temp,						
			cart03_front_temp_error 									=> m01_rs2_r1.cart03_front_temp_error,
			cart03_back_temp											=> m01_rs2_r1.cart03_back_temp,
			cart03_back_temp_error 										=> m01_rs2_r1.cart03_back_temp_error,
			cart04_front_temp											=> m01_rs2_r1.cart04_front_temp,						
			cart04_front_temp_error 									=> m01_rs2_r1.cart04_front_temp_error,
			cart04_back_temp											=> m01_rs2_r1.cart04_back_temp,
			cart04_back_temp_error 										=> m01_rs2_r1.cart04_back_temp_error,
			cart05_front_temp											=> m01_rs2_r1.cart05_front_temp,						
			cart05_front_temp_error 									=> m01_rs2_r1.cart05_front_temp_error,
			cart05_back_temp											=> m01_rs2_r1.cart05_back_temp,
			cart05_back_temp_error 										=> m01_rs2_r1.cart05_back_temp_error,
			cart06_front_temp											=> m01_rs2_r1.cart06_front_temp,						
			cart06_front_temp_error 									=> m01_rs2_r1.cart06_front_temp_error,
			cart06_back_temp											=> m01_rs2_r1.cart06_back_temp,
			cart06_back_temp_error 										=> m01_rs2_r1.cart06_back_temp_error,
			cart07_front_temp											=> m01_rs2_r1.cart07_front_temp,						
			cart07_front_temp_error 									=> m01_rs2_r1.cart07_front_temp_error,
			cart07_back_temp											=> m01_rs2_r1.cart07_back_temp,
			cart07_back_temp_error 										=> m01_rs2_r1.cart07_back_temp_error,
			cart08_front_temp											=> m01_rs2_r1.cart08_front_temp,						
			cart08_front_temp_error 									=> m01_rs2_r1.cart08_front_temp_error,
			cart08_back_temp											=> m01_rs2_r1.cart08_back_temp,
			cart08_back_temp_error 										=> m01_rs2_r1.cart08_back_temp_error,
			cart09_front_temp											=> m01_rs2_r1.cart09_front_temp,						
			cart09_front_temp_error 									=> m01_rs2_r1.cart09_front_temp_error,
			cart09_back_temp											=> m01_rs2_r1.cart09_back_temp,
			cart09_back_temp_error 										=> m01_rs2_r1.cart09_back_temp_error,
			cart10_front_temp											=> m01_rs2_r1.cart10_front_temp,						
			cart10_front_temp_error 									=> m01_rs2_r1.cart10_front_temp_error,
			cart10_back_temp											=> m01_rs2_r1.cart10_back_temp,
			cart10_back_temp_error 										=> m01_rs2_r1.cart10_back_temp_error,
			cart11_front_temp											=> m01_rs2_r1.cart11_front_temp,						
			cart11_front_temp_error 									=> m01_rs2_r1.cart11_front_temp_error,
			cart11_back_temp											=> m01_rs2_r1.cart11_back_temp,
			cart11_back_temp_error 										=> m01_rs2_r1.cart11_back_temp_error,
			cart12_front_temp											=> m01_rs2_r1.cart12_front_temp,						
			cart12_front_temp_error 									=> m01_rs2_r1.cart12_front_temp_error,
			cart12_back_temp											=> m01_rs2_r1.cart12_back_temp,
			cart12_back_temp_error 										=> m01_rs2_r1.cart12_back_temp_error,
                                                    
			inlet_co2_pump												:= m01_rs2_r1.inlet_co2_pump,
			AT_01_pump													=> m01_rs2_r1.AT_01_pump,
			inlet_co2_pump_cmd_status									=> m01_rs2_r1.inlet_co2_pump_cmd_status,
			inlet_co2_sol												:= m01_rs2_r1.inlet_co2_sol,
			AT_01_sol													=> m01_rs2_r1.AT_01_sol,
			inlet_co2_sol_cmd_status									=> m01_rs2_r1.inlet_co2_sol_cmd_status,
			outlet_co2_pump												:= m01_rs2_r1.outlet_co2_pump,
			AT_03_pump													=> m01_rs2_r1.AT_03_pump,
			outlet_co2_pump_cmd_status									=> m01_rs2_r1.outlet_co2_pump_cmd_status,
			outlet_co2_sol												:= m01_rs2_r1.outlet_co2_sol,
			AT_03_sol													=> m01_rs2_r1.AT_03_sol,
			outlet_co2_sol_cmd_status									=> m01_rs2_r1.outlet_co2_sol_cmd_status,
			repres_valve												:= m01_rs2_r1.repres_valve,
			XV_02														=> m01_rs2_r1.XV_02,
			repres_valve_open_cmd_status								=> m01_rs2_r1.repres_valve_open_cmd_status,
			repres_valve_open											:= m01_rs2_r1.repres_valve_open,
			repres_valve_closed											:= m01_rs2_r1.repres_valve_closed,
    	                                                        
			fan_vfd_control												=> m01_rs2_r1.fan_vfd_control,  		
			fan_vfd_target_vel	 		                                => m01_rs2_r1.fan_vfd_target_vel, 
			fan_vfd_enabled	 		                                    => m01_rs2_r1.fan_vfd_enabled, 
			fan_vfd_error		                                        => m01_rs2_r1.fan_vfd_error,
			fan_vfd_output												=> m01_rs2_r1.fan_vfd_output,
			fan_vfd_reset												:= m01_rs2_r1.fan_vfd_reset,
			fan_vfd_enable												:= m01_rs2_r1.fan_vfd_enable,
			fan_vfd_ecat_state											:= m01_rs2_r1.fan_vfd_ecat_state,
			fan_vfd_status												:= m01_rs2_r1.fan_vfd_status,
			fan_vfd														:= m01_rs2_r1.fan_vfd,
			fan_vfd_velocity											:= m01_rs2_r1.fan_vfd_velocity,
			fan_vfd_current												:= m01_rs2_r1.fan_vfd_current,
			fan_vfd_current_amps										=> m01_rs2_r1.fan_vfd_output_current,
			fan_vfd_temp												:= m01_rs2_r1.fan_vfd_temp,
			fan_vfd_temp_degC											=> m01_rs2_r1.fan_vfd_temperature,
			                                                    
			inlet_door_clamps_extend									:= m01_rs2_r1.inlet_door_clamps_extend,
			outlet_door_clamps_extend									:= m01_rs2_r1.outlet_door_clamps_extend,
			inlet_door_clamps_retract									:= m01_rs2_r1.inlet_door_clamps_retract,
			outlet_door_clamps_retract									:= m01_rs2_r1.outlet_door_clamps_retract,
			                                                    
			extend_clamps												:= extend_clamps,
			retract_clamps												:= retract_clamps,
			                                                    
			inlet_door_left_clamps_extend								=> m01_rs2_r1.XV_01_Left_Extend_Solenoid_Valve,
			inlet_door_right_clamps_extend								=> m01_rs2_r1.XV_01_Right_Extend_Solenoid_Valve,
			outlet_door_left_clamps_extend								=> m01_rs2_r1.XV_03_Left_Extend_Solenoid_Valve,
			outlet_door_right_clamps_extend								=> m01_rs2_r1.XV_03_Right_Extend_Solenoid_Valve,
			inlet_door_left_clamps_retract								=> m01_rs2_r1.XV_01_Left_Retract_Solenoid_Valve,
			inlet_door_right_clamps_retract								=> m01_rs2_r1.XV_01_Right_Retract_Solenoid_Valve,
			outlet_door_left_clamps_retract								=> m01_rs2_r1.XV_03_Left_Retract_Solenoid_Valve,
			outlet_door_right_clamps_retract							=> m01_rs2_r1.XV_03_Right_Retract_Solenoid_Valve,
    	                                                        
			inlet_door_left_clamps_extended								:= m01_rs2_r1.inlet_door_left_clamps_extended_ls,  
			inlet_door_right_clamps_extended							:= m01_rs2_r1.inlet_door_right_clamps_extended_ls, 
			outlet_door_left_clamps_extended							:= m01_rs2_r1.outlet_door_left_clamps_extended_ls, 
			outlet_door_right_clamps_extended							:= m01_rs2_r1.outlet_door_right_clamps_extended_ls,
			                                                    
			inlet_door_open												:= m01_rs2_r1.inlet_door_open,
			inlet_door_close											:= m01_rs2_r1.inlet_door_close,
			outlet_door_open											:= m01_rs2_r1.outlet_door_open,
			outlet_door_close											:= m01_rs2_r1.outlet_door_close,
			                                                    
			open_doors													:= open_doors,
			close_doors													:= close_doors,
			                                                    
			open_inlet_door												=> m01_rs2_r1.XV_01_Door_Open_Solenoid_Valve,
			close_inlet_door											=> m01_rs2_r1.XV_01_Door_Close_Solenoid_Valve,
			open_outlet_door											=> m01_rs2_r1.XV_03_Door_Open_Solenoid_Valve,
			close_outlet_door											=> m01_rs2_r1.XV_03_Door_Close_Solenoid_Valve,
			                                                    
			inlet_door_left_open										:= m01_rs2_r1.inlet_door_left_open_ls, 
			inlet_door_right_open										:= m01_rs2_r1.inlet_door_right_open_ls, 
			outlet_door_left_open										:= m01_rs2_r1.outlet_door_left_open_ls, 
			outlet_door_right_open										:= m01_rs2_r1.outlet_door_right_open_ls,
			inlet_door_left_closed										:= m01_rs2_r1.inlet_door_left_closed_ls, 
			inlet_door_right_closed										:= m01_rs2_r1.inlet_door_right_closed_ls, 
			outlet_door_left_closed										:= m01_rs2_r1.outlet_door_left_closed_ls, 
			outlet_door_right_closed									:= m01_rs2_r1.outlet_door_right_closed_ls,
			                                                    
			vacuum_cooling_high_temp_count								=> m01_rs2_r1.vacuum_cooling_high_temp_count,
			adsorption_high_temp_count									=> m01_rs2_r1.adsorption_high_temp_count,
			desorption_high_temp_count									=> m01_rs2_r1.desorption_air_high_temp_count);
END_ACTION

ACTION A_Reactor2_IO:
// Phase 0 - P_M01_RS02.A_Reactor2_IO
// Rev 1.0 - April 26, 2024

fb_R2_IO(	RSet														:= _RS02,
			React														:= _R2,
			
			Power_On													:= m01_rs2.power_control,
			                                                    
			sorbent_low_temp											=> m01_rs2_r2.temp_low,
			sorbent_high_temp											=> m01_rs2_r2.temp_high,
			sorbent_average_temp										=> m01_rs2_r2.temp_average,
			                                                    
			TT_01_01													:= m01_rs2_r2._01_TT_01,
			TT_01_01_offset												:= m01_rs2_r2.cart01_front_temp_offset,
			TT_01_01_error												:= m01_rs2_r2._01_TT_01_Error,
			TT_01_03													:= m01_rs2_r2._01_TT_03,               
			TT_01_03_offset												:= m01_rs2_r2.cart01_front_temp_offset,
			TT_01_03_error												:= m01_rs2_r2._01_TT_03_Error,         
			TT_02_01													:= m01_rs2_r2._02_TT_01,               
			TT_02_01_offset												:= m01_rs2_r2.cart02_front_temp_offset,
			TT_02_01_error												:= m01_rs2_r2._02_TT_01_Error,         
			TT_02_03													:= m01_rs2_r2._02_TT_03,               
			TT_02_03_offset												:= m01_rs2_r2.cart02_front_temp_offset,
			TT_02_03_error												:= m01_rs2_r2._02_TT_03_Error,         
			TT_03_01													:= m01_rs2_r2._03_TT_01,               
			TT_03_01_offset												:= m01_rs2_r2.cart03_front_temp_offset,
			TT_03_01_error												:= m01_rs2_r2._03_TT_01_Error,         
			TT_03_03													:= m01_rs2_r2._03_TT_03,               
			TT_03_03_offset												:= m01_rs2_r2.cart03_front_temp_offset,
			TT_03_03_error												:= m01_rs2_r2._03_TT_03_Error,         
			TT_04_01													:= m01_rs2_r2._04_TT_01,               
			TT_04_01_offset												:= m01_rs2_r2.cart04_front_temp_offset,
			TT_04_01_error												:= m01_rs2_r2._04_TT_01_Error,         
			TT_04_03													:= m01_rs2_r2._04_TT_03,               
			TT_04_03_offset												:= m01_rs2_r2.cart04_front_temp_offset,
			TT_04_03_error												:= m01_rs2_r2._04_TT_03_Error,         
			TT_05_01													:= m01_rs2_r2._05_TT_01,               
			TT_05_01_offset												:= m01_rs2_r2.cart05_front_temp_offset,
			TT_05_01_error												:= m01_rs2_r2._05_TT_01_Error,         
			TT_05_03													:= m01_rs2_r2._05_TT_03,               
			TT_05_03_offset												:= m01_rs2_r2.cart05_front_temp_offset,
			TT_05_03_error												:= m01_rs2_r2._05_TT_03_Error,         
			TT_06_01													:= m01_rs2_r2._06_TT_01,               
			TT_06_01_offset												:= m01_rs2_r2.cart06_front_temp_offset,
			TT_06_01_error												:= m01_rs2_r2._06_TT_01_Error,         
			TT_06_03													:= m01_rs2_r2._06_TT_03,               
			TT_06_03_offset												:= m01_rs2_r2.cart06_front_temp_offset,
			TT_06_03_error												:= m01_rs2_r2._06_TT_03_Error,         
			TT_07_01													:= m01_rs2_r2._07_TT_01,               
			TT_07_01_offset												:= m01_rs2_r2.cart07_front_temp_offset,
			TT_07_01_error												:= m01_rs2_r2._07_TT_01_Error,         
			TT_07_03													:= m01_rs2_r2._07_TT_03,               
			TT_07_03_offset												:= m01_rs2_r2.cart07_front_temp_offset,
			TT_07_03_error												:= m01_rs2_r2._07_TT_03_Error,         
			TT_08_01													:= m01_rs2_r2._08_TT_01,               
			TT_08_01_offset												:= m01_rs2_r2.cart08_front_temp_offset,
			TT_08_01_error												:= m01_rs2_r2._08_TT_01_Error,         
			TT_08_03													:= m01_rs2_r2._08_TT_03,               
			TT_08_03_offset												:= m01_rs2_r2.cart08_front_temp_offset,
			TT_08_03_error												:= m01_rs2_r2._08_TT_03_Error,         
			TT_09_01													:= m01_rs2_r2._09_TT_01,               
			TT_09_01_offset												:= m01_rs2_r2.cart09_front_temp_offset,
			TT_09_01_error												:= m01_rs2_r2._09_TT_01_Error,         
			TT_09_03													:= m01_rs2_r2._09_TT_03,               
			TT_09_03_offset												:= m01_rs2_r2.cart09_front_temp_offset,
			TT_09_03_error												:= m01_rs2_r2._09_TT_03_Error,         
			TT_10_01													:= m01_rs2_r2._10_TT_01,               
			TT_10_01_offset												:= m01_rs2_r2.cart10_front_temp_offset,
			TT_10_01_error												:= m01_rs2_r2._10_TT_01_Error,         
			TT_10_03													:= m01_rs2_r2._10_TT_03,               
			TT_10_03_offset												:= m01_rs2_r2.cart10_front_temp_offset,
			TT_10_03_error												:= m01_rs2_r2._10_TT_03_Error,         
			TT_11_01													:= m01_rs2_r2._11_TT_01,               
			TT_11_01_offset												:= m01_rs2_r2.cart11_front_temp_offset,
			TT_11_01_error												:= m01_rs2_r2._11_TT_01_Error,         
			TT_11_03													:= m01_rs2_r2._11_TT_03,               
			TT_11_03_offset												:= m01_rs2_r2.cart11_front_temp_offset,
			TT_11_03_error												:= m01_rs2_r2._11_TT_03_Error,         
			TT_12_01													:= m01_rs2_r2._12_TT_01,               
			TT_12_01_offset												:= m01_rs2_r2.cart12_front_temp_offset,
			TT_12_01_error												:= m01_rs2_r2._12_TT_01_Error,         
			TT_12_03													:= m01_rs2_r2._12_TT_03,               
			TT_12_03_offset												:= m01_rs2_r2.cart12_front_temp_offset,
			TT_12_03_error												:= m01_rs2_r2._12_TT_03_Error,         

